QRS_NEXT_CUT()
PTP {E1 36177.176,E2 36177.176}
PTP {X 0,Y 759.945,A -85,B 0,C 180,E1 36177.176,E2 36177.176,E3 0,E4 0,E5 0,E6 0}
QRS_SPEED_INIT()
LIN {X 0,Y 759.945,Z 1215,A -85,B 0,C 180,E1 36177.176,E2 36177.176,E3 0,E4 0,E5 0,E6 0} C_VEL
LIN {X 0,Y 759.945,Z 319.648,A -85,B 0,C 180,E1 36177.176,E2 36177.176} C_VEL
LIN {X 0,Y 759.945,Z 311.576,A -85,B 0,C 180,E1 36177.176,E2 36177.176} C_VEL
LIN {X 0,Y 759.914,Z 309.576,A -85,B 0,C 180,E1 36177.025,E2 36177.025} C_VEL
LIN {X 0,Y 759.839,Z 309.574,A -85,B 0,C 180,E1 36174.336,E2 36174.336} C_VEL
LIN {X 0,Y 759.839,Z 309.572,A -85,B 0,C 180,E1 36171.906,E2 36171.906} C_VEL
LIN {X 0,Y 759.916,Z 309.571,A -85,B 0,C 180,E1 36169.155,E2 36169.155} C_VEL
LIN {X 0,Y 759.839,Z 309.575,A -85,B 0,C 180,E1 36166.298,E2 36166.298} C_VEL
LIN {X 0,Y 759.826,Z 309.574,A -85,B 0,C 180,E1 36163.957,E2 36163.957} C_VEL
LIN {X 0,Y 759.829,Z 309.574,A -85,B 0,C 180,E1 36161.669,E2 36161.669} C_VEL
LIN {X 0,Y 759.912,Z 309.571,A -85,B 0,C 180,E1 36158.948,E2 36158.948} C_VEL
LIN {X 0,Y 759.831,Z 309.576,A -85,B 0,C 180,E1 36156.089,E2 36156.089} C_VEL
LIN {X 0,Y 759.817,Z 309.575,A -85,B 0,C 180,E1 36153.825,E2 36153.825} C_VEL
LIN {X 0,Y 759.814,Z 309.576,A -85,B 0,C 180,E1 36151.551,E2 36151.551} C_VEL
LIN {X 0,Y 759.828,Z 309.575,A -85,B 0,C 180,E1 36149.209,E2 36149.209} C_VEL
LIN {X 0,Y 759.89,Z 309.576,A -85,B 0,C 180,E1 36146.36,E2 36146.36} C_VEL
LIN {X 0,Y 759.815,Z 309.577,A -85,B 0,C 180,E1 36143.771,E2 36143.771} C_VEL
LIN {X 0,Y 759.802,Z 309.576,A -85,B 0,C 180,E1 36141.504,E2 36141.504} C_VEL
LIN {X 0,Y 759.801,Z 309.578,A -85,B 0,C 180,E1 36139.252,E2 36139.252} C_VEL
LIN {X 0,Y 759.811,Z 309.578,A -85,B 0,C 180,E1 36137.025,E2 36137.025} C_VEL
LIN {X 0,Y 759.909,Z 309.578,A -85,B 0,C 180,E1 36134.291,E2 36134.291} C_VEL
LIN {X 0,Y 759.83,Z 309.76,A -85,B 0,C 180,E1 36131.629,E2 36131.629} C_VEL
LIN {X 0,Y 759.819,Z 321.429,A -85,B 0,C 180,E1 36130.869,E2 36130.869} C_VEL
LIN {X 0,Y 759.897,Z 497.056,A -85,B 0,C 180,E1 36128.746,E2 36128.746} C_VEL
LIN {X 0,Y 759.916,Z 717.097,A -85,B 0,C 180,E1 36126.177,E2 36126.177} C_VEL
LIN {X 0,Y 759.91,Z 798.77,A -85,B 0,C 180,E1 36125.223,E2 36125.223} C_VEL
LIN {X 0,Y 759.911,Z 825.377,A -85,B 0,C 180,E1 36124.77,E2 36124.77} C_VEL
LIN {X 0,Y 759.914,Z 852.595,A -85,B 0,C 180,E1 36124.143,E2 36124.143} C_VEL
LIN {X 0,Y 759.907,Z 874.72,A -85,B 0,C 180,E1 36123.506,E2 36123.506} C_VEL
LIN {X 0,Y 759.919,Z 892.583,A -85,B 0,C 180,E1 36122.915,E2 36122.915} C_VEL
LIN {X 0,Y 759.919,Z 911.329,A -85,B 0,C 180,E1 36122.215,E2 36122.215} C_VEL
LIN {X 0,Y 759.913,Z 929.676,A -85,B 0,C 180,E1 36121.446,E2 36121.446} C_VEL
LIN {X 0,Y 759.915,Z 948.5,A -85,B 0,C 180,E1 36120.566,E2 36120.566} C_VEL
LIN {X 0,Y 759.911,Z 966.95,A -85,B 0,C 180,E1 36119.611,E2 36119.611} C_VEL
LIN {X 0,Y 759.909,Z 986.655,A -85,B 0,C 180,E1 36118.483,E2 36118.483} C_VEL
LIN {X 0,Y 759.91,Z 1010.382,A -85,B 0,C 180,E1 36116.954,E2 36116.954} C_VEL
LIN {X 0,Y 759.915,Z 1028.464,A -85,B 0,C 180,E1 36115.65,E2 36115.65} C_VEL
LIN {X 0,Y 759.893,Z 1046.844,A -85,B 0,C 180,E1 36114.195,E2 36114.195} C_VEL
LIN {X 0,Y 759.92,Z 1065.796,A -85,B 0,C 180,E1 36112.512,E2 36112.512} C_VEL
LIN {X 0,Y 759.897,Z 1080.62,A -85,B 0,C 180,E1 36111.052,E2 36111.052} C_VEL
LIN {X 0,Y 759.914,Z 1094.69,A -85,B 0,C 180,E1 36109.524,E2 36109.524} C_VEL
LIN {X 0,Y 759.9,Z 1109.841,A -85,B 0,C 180,E1 36107.695,E2 36107.695} C_VEL
LIN {X 0,Y 759.89,Z 1122.953,A -85,B 0,C 180,E1 36105.871,E2 36105.871} C_VEL
LIN {X 0,Y 759.917,Z 1132.856,A -85,B 0,C 180,E1 36104.321,E2 36104.321} C_VEL
LIN {X 0,Y 759.908,Z 1141.641,A -85,B 0,C 180,E1 36102.771,E2 36102.771} C_VEL
LIN {X 0,Y 759.903,Z 1149.647,A -85,B 0,C 180,E1 36101.152,E2 36101.152} C_VEL
LIN {X 0,Y 759.916,Z 1157.473,A -85,B 0,C 180,E1 36099.303,E2 36099.303} C_VEL
LIN {X 0,Y 759.91,Z 1164.123,A -85,B 0,C 180,E1 36097.333,E2 36097.333} C_VEL
LIN {X 0,Y 759.906,Z 1169.35,A -85,B 0,C 180,E1 36095.285,E2 36095.285} C_VEL
LIN {X 0,Y 759.909,Z 1172.83,A -85,B 0,C 180,E1 36093.243,E2 36093.243} C_VEL
LIN {X 0,Y 759.911,Z 1174.612,A -85,B 0,C 180,E1 36091.282,E2 36091.282} C_VEL
LIN {X 0,Y 759.889,Z 1174.863,A -85,B 0,C 180,E1 36089.472,E2 36089.472} C_VEL
LIN {X 0,Y 759.907,Z 1173.954,A -85,B 0,C 180,E1 36087.662,E2 36087.662} C_VEL
LIN {X 0,Y 759.909,Z 1171.128,A -85,B 0,C 180,E1 36085.548,E2 36085.548} C_VEL
LIN {X 0,Y 759.918,Z 1166.878,A -85,B 0,C 180,E1 36083.579,E2 36083.579} C_VEL
LIN {X 0,Y 759.916,Z 1160.788,A -85,B 0,C 180,E1 36081.526,E2 36081.526} C_VEL
LIN {X 0,Y 759.893,Z 1152.605,A -85,B 0,C 180,E1 36079.399,E2 36079.399} C_VEL
LIN {X 0,Y 759.913,Z 1142.939,A -85,B 0,C 180,E1 36077.384,E2 36077.384} C_VEL
LIN {X 0,Y 759.918,Z 1133.86,A -85,B 0,C 180,E1 36075.756,E2 36075.756} C_VEL
LIN {X 0,Y 759.894,Z 1123.989,A -85,B 0,C 180,E1 36074.195,E2 36074.195} C_VEL
LIN {X 0,Y 759.908,Z 1112.833,A -85,B 0,C 180,E1 36072.622,E2 36072.622} C_VEL
LIN {X 0,Y 759.912,Z 1097.622,A -85,B 0,C 180,E1 36070.716,E2 36070.716} C_VEL
LIN {X 0,Y 759.893,Z 1082.269,A -85,B 0,C 180,E1 36069.029,E2 36069.029} C_VEL
LIN {X 0,Y 759.903,Z 1067.592,A -85,B 0,C 180,E1 36067.569,E2 36067.569} C_VEL
LIN {X 0,Y 759.892,Z 1048.945,A -85,B 0,C 180,E1 36065.886,E2 36065.886} C_VEL
LIN {X 0,Y 759.917,Z 1029.425,A -85,B 0,C 180,E1 36064.332,E2 36064.332} C_VEL
LIN {X 0,Y 759.91,Z 1012.274,A -85,B 0,C 180,E1 36063.088,E2 36063.088} C_VEL
LIN {X 0,Y 759.915,Z 990.289,A -85,B 0,C 180,E1 36061.642,E2 36061.642} C_VEL
LIN {X 0,Y 759.908,Z 967.865,A -85,B 0,C 180,E1 36060.348,E2 36060.348} C_VEL
LIN {X 0,Y 759.917,Z 949.16,A -85,B 0,C 180,E1 36059.376,E2 36059.376} C_VEL
LIN {X 0,Y 759.913,Z 930.486,A -85,B 0,C 180,E1 36058.5,E2 36058.5} C_VEL
LIN {X 0,Y 759.919,Z 911.728,A -85,B 0,C 180,E1 36057.711,E2 36057.711} C_VEL
LIN {X 0,Y 759.92,Z 893.856,A -85,B 0,C 180,E1 36057.04,E2 36057.04} C_VEL
LIN {X 0,Y 759.909,Z 875.417,A -85,B 0,C 180,E1 36056.426,E2 36056.426} C_VEL
LIN {X 0,Y 759.912,Z 853.71,A -85,B 0,C 180,E1 36055.795,E2 36055.795} C_VEL
LIN {X 0,Y 759.914,Z 826.054,A -85,B 0,C 180,E1 36055.155,E2 36055.155} C_VEL
LIN {X 0,Y 759.91,Z 799.959,A -85,B 0,C 180,E1 36054.704,E2 36054.704} C_VEL
LIN {X 0,Y 759.919,Z 743.099,A -85,B 0,C 180,E1 36054.031,E2 36054.031} C_VEL
LIN {X 0,Y 759.91,Z 519.207,A -85,B 0,C 180,E1 36051.428,E2 36051.428} C_VEL
LIN {X 0,Y 759.834,Z 329.757,A -85,B 0,C 180,E1 36049.144,E2 36049.144} C_VEL
LIN {X 0,Y 759.825,Z 320.904,A -85,B 0,C 180,E1 36049.031,E2 36049.031} C_VEL
LIN {X 0,Y 759.848,Z 309.579,A -85,B 0,C 180,E1 36048.254,E2 36048.254} C_VEL
LIN {X 0,Y 759.842,Z 309.577,A -85,B 0,C 180,E1 36045.177,E2 36045.177} C_VEL
LIN {X 0,Y 759.817,Z 309.577,A -85,B 0,C 180,E1 36042.864,E2 36042.864} C_VEL
LIN {X 0,Y 759.808,Z 309.577,A -85,B 0,C 180,E1 36040.648,E2 36040.648} C_VEL
LIN {X 0,Y 759.805,Z 309.577,A -85,B 0,C 180,E1 36038.466,E2 36038.466} C_VEL
LIN {X 0,Y 759.82,Z 309.577,A -85,B 0,C 180,E1 36036.102,E2 36036.102} C_VEL
LIN {X 0,Y 759.886,Z 309.578,A -85,B 0,C 180,E1 36033.279,E2 36033.279} C_VEL
LIN {X 0,Y 759.815,Z 309.576,A -85,B 0,C 180,E1 36030.704,E2 36030.704} C_VEL
LIN {X 0,Y 759.807,Z 309.577,A -85,B 0,C 180,E1 36028.45,E2 36028.45} C_VEL
LIN {X 0,Y 759.807,Z 309.576,A -85,B 0,C 180,E1 36026.243,E2 36026.243} C_VEL
LIN {X 0,Y 759.814,Z 309.576,A -85,B 0,C 180,E1 36024.042,E2 36024.042} C_VEL
LIN {X 0,Y 759.862,Z 309.577,A -85,B 0,C 180,E1 36021.519,E2 36021.519} C_VEL
LIN {X 0,Y 759.844,Z 309.574,A -85,B 0,C 180,E1 36018.569,E2 36018.569} C_VEL
LIN {X 0,Y 759.822,Z 309.574,A -85,B 0,C 180,E1 36016.2,E2 36016.2} C_VEL
LIN {X 0,Y 759.822,Z 309.574,A -85,B 0,C 180,E1 36013.935,E2 36013.935} C_VEL
LIN {X 0,Y 759.843,Z 309.576,A -85,B 0,C 180,E1 36011.538,E2 36011.538} C_VEL
LIN {X 0,Y 759.897,Z 309.571,A -85,B 0,C 180,E1 36008.627,E2 36008.627} C_VEL
LIN {X 0,Y 759.837,Z 309.573,A -85,B 0,C 180,E1 36006.043,E2 36006.043} C_VEL
LIN {X 0,Y 759.833,Z 309.573,A -85,B 0,C 180,E1 36003.697,E2 36003.697} C_VEL
LIN {X 0,Y 759.865,Z 309.575,A -85,B 0,C 180,E1 36001.206,E2 36001.206} C_VEL
LIN {X 0,Y 759.867,Z 309.57,A -85,B 0,C 180,E1 35998.115,E2 35998.115} C_VEL
LIN {X 0,Y 759.842,Z 309.572,A -85,B 0,C 180,E1 35995.623,E2 35995.623} C_VEL
LIN {X 0,Y 759.863,Z 309.575,A -85,B 0,C 180,E1 35993.123,E2 35993.123} C_VEL
LIN {X 0,Y 759.906,Z 309.567,A -85,B 0,C 180,E1 35990.151,E2 35990.151} C_VEL
LIN {X 0,Y 759.85,Z 309.572,A -85,B 0,C 180,E1 35987.46,E2 35987.46} C_VEL
LIN {X 0,Y 759.875,Z 309.574,A -85,B 0,C 180,E1 35984.898,E2 35984.898} C_VEL
LIN {X 0,Y 759.904,Z 309.567,A -85,B 0,C 180,E1 35981.909,E2 35981.909} C_VEL
LIN {X 0,Y 759.858,Z 309.57,A -85,B 0,C 180,E1 35979.269,E2 35979.269} C_VEL
LIN {X 0,Y 759.895,Z 309.577,A -85,B 0,C 180,E1 35976.585,E2 35976.585} C_VEL
LIN {X 0,Y 759.894,Z 309.566,A -85,B 0,C 180,E1 35973.593,E2 35973.593} C_VEL
LIN {X 0,Y 759.867,Z 309.572,A -85,B 0,C 180,E1 35970.864,E2 35970.864} C_VEL
LIN {X 0,Y 759.911,Z 309.575,A -85,B 0,C 180,E1 35968.154,E2 35968.154} C_VEL
LIN {X 0,Y 759.887,Z 309.567,A -85,B 0,C 180,E1 35965.266,E2 35965.266} C_VEL
LIN {X 0,Y 759.887,Z 309.574,A -85,B 0,C 180,E1 35962.466,E2 35962.466} C_VEL
LIN {X 0,Y 759.91,Z 309.566,A -85,B 0,C 180,E1 35959.509,E2 35959.509} C_VEL
LIN {X 0,Y 759.876,Z 309.571,A -85,B 0,C 180,E1 35956.72,E2 35956.72} C_VEL
LIN {X 0,Y 759.913,Z 309.577,A -85,B 0,C 180,E1 35953.967,E2 35953.967} C_VEL
LIN {X 0,Y 759.9,Z 309.834,A -85,B 0,C 180,E1 35953.53,E2 35953.53} C_VEL
LIN {X 0,Y 759.904,Z 350.585,A -85,B 0,C 180,E1 35950.919,E2 35950.919} C_VEL
LIN {X 0,Y 759.912,Z 566.438,A -85,B 0,C 180,E1 35948.324,E2 35948.324} C_VEL
LIN {X 0,Y 759.917,Z 792.185,A -85,B 0,C 180,E1 35945.706,E2 35945.706} C_VEL
LIN {X 0,Y 759.911,Z 831.844,A -85,B 0,C 180,E1 35945.223,E2 35945.223} C_VEL
LIN {X 0,Y 759.908,Z 857.526,A -85,B 0,C 180,E1 35944.77,E2 35944.77} C_VEL
LIN {X 0,Y 759.913,Z 884.353,A -85,B 0,C 180,E1 35944.143,E2 35944.143} C_VEL
LIN {X 0,Y 759.907,Z 909.243,A -85,B 0,C 180,E1 35943.411,E2 35943.411} C_VEL
LIN {X 0,Y 759.918,Z 937.245,A -85,B 0,C 180,E1 35942.423,E2 35942.423} C_VEL
LIN {X 0,Y 759.915,Z 958.588,A -85,B 0,C 180,E1 35941.539,E2 35941.539} C_VEL
LIN {X 0,Y 759.912,Z 977.503,A -85,B 0,C 180,E1 35940.661,E2 35940.661} C_VEL
LIN {X 0,Y 759.913,Z 995.702,A -85,B 0,C 180,E1 35939.723,E2 35939.723} C_VEL
LIN {X 0,Y 759.909,Z 1013.707,A -85,B 0,C 180,E1 35938.702,E2 35938.702} C_VEL
LIN {X 0,Y 759.911,Z 1035.516,A -85,B 0,C 180,E1 35937.335,E2 35937.335} C_VEL
LIN {X 0,Y 759.912,Z 1056.845,A -85,B 0,C 180,E1 35935.818,E2 35935.818} C_VEL
LIN {X 0,Y 759.91,Z 1073.823,A -85,B 0,C 180,E1 35934.485,E2 35934.485} C_VEL
LIN {X 0,Y 759.901,Z 1092.853,A -85,B 0,C 180,E1 35932.84,E2 35932.84} C_VEL
LIN {X 0,Y 759.895,Z 1109.495,A -85,B 0,C 180,E1 35931.213,E2 35931.213} C_VEL
LIN {X 0,Y 759.905,Z 1122.958,A -85,B 0,C 180,E1 35929.764,E2 35929.764} C_VEL
LIN {X 0,Y 759.897,Z 1135.732,A -85,B 0,C 180,E1 35928.249,E2 35928.249} C_VEL
LIN {X 0,Y 759.909,Z 1150.031,A -85,B 0,C 180,E1 35926.354,E2 35926.354} C_VEL
LIN {X 0,Y 759.909,Z 1162.194,A -85,B 0,C 180,E1 35924.477,E2 35924.477} C_VEL
LIN {X 0,Y 759.91,Z 1171.058,A -85,B 0,C 180,E1 35922.925,E2 35922.925} C_VEL
LIN {X 0,Y 759.91,Z 1178.784,A -85,B 0,C 180,E1 35921.383,E2 35921.383} C_VEL
LIN {X 0,Y 759.906,Z 1186.43,A -85,B 0,C 180,E1 35919.619,E2 35919.619} C_VEL
LIN {X 0,Y 759.908,Z 1193.594,A -85,B 0,C 180,E1 35917.561,E2 35917.561} C_VEL
LIN {X 0,Y 759.91,Z 1199.108,A -85,B 0,C 180,E1 35915.436,E2 35915.436} C_VEL
LIN {X 0,Y 759.916,Z 1202.585,A -85,B 0,C 180,E1 35913.47,E2 35913.47} C_VEL
LIN {X 0,Y 759.914,Z 1204.58,A -85,B 0,C 180,E1 35911.432,E2 35911.432} C_VEL
LIN {X 0,Y 759.889,Z 1204.849,A -85,B 0,C 180,E1 35909.472,E2 35909.472} C_VEL
LIN {X 0,Y 759.907,Z 1203.907,A -85,B 0,C 180,E1 35907.662,E2 35907.662} C_VEL
LIN {X 0,Y 759.908,Z 1201.054,A -85,B 0,C 180,E1 35905.548,E2 35905.548} C_VEL
LIN {X 0,Y 759.914,Z 1196.566,A -85,B 0,C 180,E1 35903.503,E2 35903.503} C_VEL
LIN {X 0,Y 759.913,Z 1190.629,A -85,B 0,C 180,E1 35901.526,E2 35901.526} C_VEL
LIN {X 0,Y 759.896,Z 1182.68,A -85,B 0,C 180,E1 35899.462,E2 35899.462} C_VEL
LIN {X 0,Y 759.905,Z 1173.111,A -85,B 0,C 180,E1 35897.461,E2 35897.461} C_VEL
LIN {X 0,Y 759.91,Z 1164.056,A -85,B 0,C 180,E1 35895.834,E2 35895.834} C_VEL
LIN {X 0,Y 759.894,Z 1154.212,A -85,B 0,C 180,E1 35894.273,E2 35894.273} C_VEL
LIN {X 0,Y 759.904,Z 1143.666,A -85,B 0,C 180,E1 35892.78,E2 35892.78} C_VEL
LIN {X 0,Y 759.896,Z 1130.456,A -85,B 0,C 180,E1 35891.1,E2 35891.1} C_VEL
LIN {X 0,Y 759.898,Z 1113.394,A -85,B 0,C 180,E1 35889.191,E2 35889.191} C_VEL
LIN {X 0,Y 759.898,Z 1098.828,A -85,B 0,C 180,E1 35887.732,E2 35887.732} C_VEL
LIN {X 0,Y 759.911,Z 1082.654,A -85,B 0,C 180,E1 35886.258,E2 35886.258} C_VEL
LIN {X 0,Y 759.91,Z 1061.274,A -85,B 0,C 180,E1 35884.516,E2 35884.516} C_VEL
LIN {X 0,Y 759.91,Z 1044.049,A -85,B 0,C 180,E1 35883.257,E2 35883.257} C_VEL
LIN {X 0,Y 759.914,Z 1026.242,A -85,B 0,C 180,E1 35882.069,E2 35882.069} C_VEL
LIN {X 0,Y 759.905,Z 1003.454,A -85,B 0,C 180,E1 35880.695,E2 35880.695} C_VEL
LIN {X 0,Y 759.916,Z 981.266,A -85,B 0,C 180,E1 35879.525,E2 35879.525} C_VEL
LIN {X 0,Y 759.912,Z 961.681,A -85,B 0,C 180,E1 35878.598,E2 35878.598} C_VEL
LIN {X 0,Y 759.918,Z 942.461,A -85,B 0,C 180,E1 35877.785,E2 35877.785} C_VEL
LIN {X 0,Y 759.919,Z 923.853,A -85,B 0,C 180,E1 35877.085,E2 35877.085} C_VEL
LIN {X 0,Y 759.909,Z 905.51,A -85,B 0,C 180,E1 35876.474,E2 35876.474} C_VEL
LIN {X 0,Y 759.913,Z 882.835,A -85,B 0,C 180,E1 35875.818,E2 35875.818} C_VEL
LIN {X 0,Y 759.911,Z 855.67,A -85,B 0,C 180,E1 35875.191,E2 35875.191} C_VEL
LIN {X 0,Y 759.91,Z 829.101,A -85,B 0,C 180,E1 35874.737,E2 35874.737} C_VEL
LIN {X 0,Y 759.915,Z 735.994,A -85,B 0,C 180,E1 35873.651,E2 35873.651} C_VEL
LIN {X 0,Y 759.912,Z 513.174,A -85,B 0,C 180,E1 35871.045,E2 35871.045} C_VEL
LIN {X 0,Y 759.904,Z 350.467,A -85,B 0,C 180,E1 35869.074,E2 35869.074} C_VEL
LIN {X 0,Y 759.9,Z 309.834,A -85,B 0,C 180,E1 35866.47,E2 35866.47} C_VEL
LIN {X 0,Y 759.913,Z 309.577,A -85,B 0,C 180,E1 35866.033,E2 35866.033} C_VEL
LIN {X 0,Y 759.877,Z 309.57,A -85,B 0,C 180,E1 35863.201,E2 35863.201} C_VEL
LIN {X 0,Y 759.907,Z 309.566,A -85,B 0,C 180,E1 35860.443,E2 35860.443} C_VEL
LIN {X 0,Y 759.887,Z 309.575,A -85,B 0,C 180,E1 35857.534,E2 35857.534} C_VEL
LIN {X 0,Y 759.892,Z 309.566,A -85,B 0,C 180,E1 35854.678,E2 35854.678} C_VEL
LIN {X 0,Y 759.908,Z 309.578,A -85,B 0,C 180,E1 35851.669,E2 35851.669} C_VEL
LIN {X 0,Y 759.865,Z 309.571,A -85,B 0,C 180,E1 35848.952,E2 35848.952} C_VEL
LIN {X 0,Y 759.911,Z 309.566,A -85,B 0,C 180,E1 35846.189,E2 35846.189} C_VEL
LIN {X 0,Y 759.882,Z 309.575,A -85,B 0,C 180,E1 35843.251,E2 35843.251} C_VEL
LIN {X 0,Y 759.864,Z 309.569,A -85,B 0,C 180,E1 35840.569,E2 35840.569} C_VEL
LIN {X 0,Y 759.91,Z 309.57,A -85,B 0,C 180,E1 35837.774,E2 35837.774} C_VEL
LIN {X 0,Y 759.865,Z 309.573,A -85,B 0,C 180,E1 35834.946,E2 35834.946} C_VEL
LIN {X 0,Y 759.862,Z 309.57,A -85,B 0,C 180,E1 35832.308,E2 35832.308} C_VEL
LIN {X 0,Y 759.913,Z 309.573,A -85,B 0,C 180,E1 35829.467,E2 35829.467} C_VEL
LIN {X 0,Y 759.856,Z 309.574,A -85,B 0,C 180,E1 35826.726,E2 35826.726} C_VEL
LIN {X 0,Y 759.849,Z 309.571,A -85,B 0,C 180,E1 35824.226,E2 35824.226} C_VEL
LIN {X 0,Y 759.915,Z 309.568,A -85,B 0,C 180,E1 35821.508,E2 35821.508} C_VEL
LIN {X 0,Y 759.856,Z 309.574,A -85,B 0,C 180,E1 35818.643,E2 35818.643} C_VEL
LIN {X 0,Y 759.914,Z 309.576,A -85,B 0,C 180,E1 35817.025,E2 35817.025} C_VEL
LIN {X 0,Y 758.859,Z 309.699,A -85,B 0,C 180,E1 35816.444,E2 35816.444} C_VEL
LIN {X 0,Y 752.447,Z 310.504,A -85,B 0,C 180,E1 35814.818,E2 35814.818} C_VEL
LIN {X 0,Y 751.904,Z 310.564,A -85,B 0,C 180,E1 35814.396,E2 35814.396} C_VEL
LIN {X 0,Y 751.897,Z 310.561,A -85,B 0,C 180,E1 35811.973,E2 35811.973} C_VEL
LIN {X 0,Y 751.966,Z 310.558,A -85,B 0,C 180,E1 35809.271,E2 35809.271} C_VEL
LIN {X 0,Y 751.908,Z 310.563,A -85,B 0,C 180,E1 35806.386,E2 35806.386} C_VEL
LIN {X 0,Y 751.888,Z 310.563,A -85,B 0,C 180,E1 35804.021,E2 35804.021} C_VEL
LIN {X 0,Y 751.889,Z 310.563,A -85,B 0,C 180,E1 35801.708,E2 35801.708} C_VEL
LIN {X 0,Y 751.955,Z 310.559,A -85,B 0,C 180,E1 35799.041,E2 35799.041} C_VEL
LIN {X 0,Y 751.898,Z 310.565,A -85,B 0,C 180,E1 35796.155,E2 35796.155} C_VEL
LIN {X 0,Y 751.877,Z 310.564,A -85,B 0,C 180,E1 35793.799,E2 35793.799} C_VEL
LIN {X 0,Y 751.876,Z 310.565,A -85,B 0,C 180,E1 35791.523,E2 35791.523} C_VEL
LIN {X 0,Y 751.898,Z 310.562,A -85,B 0,C 180,E1 35789.115,E2 35789.115} C_VEL
LIN {X 0,Y 751.9,Z 310.564,A -85,B 0,C 180,E1 35786.046,E2 35786.046} C_VEL
LIN {X 0,Y 751.871,Z 310.567,A -85,B 0,C 180,E1 35783.695,E2 35783.695} C_VEL
LIN {X 0,Y 751.862,Z 310.564,A -85,B 0,C 180,E1 35781.439,E2 35781.439} C_VEL
LIN {X 0,Y 751.867,Z 310.567,A -85,B 0,C 180,E1 35779.133,E2 35779.133} C_VEL
LIN {X 0,Y 751.93,Z 310.567,A -85,B 0,C 180,E1 35776.554,E2 35776.554} C_VEL
LIN {X 0,Y 751.886,Z 310.569,A -85,B 0,C 180,E1 35773.643,E2 35773.643} C_VEL
LIN {X 0,Y 751.978,Z 310.677,A -85,B 0,C 180,E1 35772.101,E2 35772.101} C_VEL
LIN {X 0,Y 753.147,Z 314.7,A -85,B 0,C 180,E1 35771.744,E2 35771.744} C_VEL
LIN {X 0,Y 753.251,Z 321.517,A -85,B 0,C 180,E1 35771.302,E2 35771.302} C_VEL
LIN {X 0,Y 753.757,Z 324.477,A -85,B 0,C 180,E1 35771.232,E2 35771.232} C_VEL
LIN {X 0,Y 753.644,Z 503.901,A -85,B 0,C 180,E1 35769.047,E2 35769.047} C_VEL
LIN {X 0,Y 753.443,Z 729.229,A -85,B 0,C 180,E1 35766.397,E2 35766.397} C_VEL
LIN {X 0,Y 753.353,Z 799.594,A -85,B 0,C 180,E1 35765.564,E2 35765.564} C_VEL
LIN {X 0,Y 753.277,Z 826.438,A -85,B 0,C 180,E1 35765.099,E2 35765.099} C_VEL
LIN {X 0,Y 753.196,Z 853.912,A -85,B 0,C 180,E1 35764.457,E2 35764.457} C_VEL
LIN {X 0,Y 753.096,Z 877.658,A -85,B 0,C 180,E1 35763.758,E2 35763.758} C_VEL
LIN {X 0,Y 753.006,Z 902.747,A -85,B 0,C 180,E1 35762.893,E2 35762.893} C_VEL
LIN {X 0,Y 752.86,Z 927.706,A -85,B 0,C 180,E1 35761.864,E2 35761.864} C_VEL
LIN {X 0,Y 752.761,Z 947.625,A -85,B 0,C 180,E1 35760.933,E2 35760.933} C_VEL
LIN {X 0,Y 752.667,Z 966.211,A -85,B 0,C 180,E1 35759.966,E2 35759.966} C_VEL
LIN {X 0,Y 752.574,Z 984.97,A -85,B 0,C 180,E1 35758.888,E2 35758.888} C_VEL
LIN {X 0,Y 752.438,Z 1007.964,A -85,B 0,C 180,E1 35757.416,E2 35757.416} C_VEL
LIN {X 0,Y 752.339,Z 1027.364,A -85,B 0,C 180,E1 35756.013,E2 35756.013} C_VEL
LIN {X 0,Y 752.28,Z 1044.293,A -85,B 0,C 180,E1 35754.667,E2 35754.667} C_VEL
LIN {X 0,Y 752.173,Z 1063.244,A -85,B 0,C 180,E1 35753.005,E2 35753.005} C_VEL
LIN {X 0,Y 752.11,Z 1079.847,A -85,B 0,C 180,E1 35751.362,E2 35751.362} C_VEL
LIN {X 0,Y 752.054,Z 1093.276,A -85,B 0,C 180,E1 35749.898,E2 35749.898} C_VEL
LIN {X 0,Y 752.028,Z 1106.421,A -85,B 0,C 180,E1 35748.317,E2 35748.317} C_VEL
LIN {X 0,Y 751.966,Z 1121.591,A -85,B 0,C 180,E1 35746.25,E2 35746.25} C_VEL
LIN {X 0,Y 751.955,Z 1132.578,A -85,B 0,C 180,E1 35744.524,E2 35744.524} C_VEL
LIN {X 0,Y 751.926,Z 1141.644,A -85,B 0,C 180,E1 35742.908,E2 35742.908} C_VEL
LIN {X 0,Y 751.93,Z 1149.293,A -85,B 0,C 180,E1 35741.35,E2 35741.35} C_VEL
LIN {X 0,Y 751.915,Z 1156.846,A -85,B 0,C 180,E1 35739.568,E2 35739.568} C_VEL
LIN {X 0,Y 751.912,Z 1163.685,A -85,B 0,C 180,E1 35737.565,E2 35737.565} C_VEL
LIN {X 0,Y 751.909,Z 1169.179,A -85,B 0,C 180,E1 35735.418,E2 35735.418} C_VEL
LIN {X 0,Y 751.91,Z 1172.729,A -85,B 0,C 180,E1 35733.354,E2 35733.354} C_VEL
LIN {X 0,Y 751.912,Z 1174.589,A -85,B 0,C 180,E1 35731.372,E2 35731.372} C_VEL
LIN {X 0,Y 751.889,Z 1174.863,A -85,B 0,C 180,E1 35729.467,E2 35729.467} C_VEL
LIN {X 0,Y 751.907,Z 1173.953,A -85,B 0,C 180,E1 35727.637,E2 35727.637} C_VEL
LIN {X 0,Y 751.907,Z 1171.127,A -85,B 0,C 180,E1 35725.5,E2 35725.5} C_VEL
LIN {X 0,Y 751.917,Z 1166.876,A -85,B 0,C 180,E1 35723.51,E2 35723.51} C_VEL
LIN {X 0,Y 751.923,Z 1160.786,A -85,B 0,C 180,E1 35721.435,E2 35721.435} C_VEL
LIN {X 0,Y 751.904,Z 1152.823,A -85,B 0,C 180,E1 35719.338,E2 35719.338} C_VEL
LIN {X 0,Y 751.941,Z 1143.349,A -85,B 0,C 180,E1 35717.326,E2 35717.326} C_VEL
LIN {X 0,Y 751.961,Z 1134.324,A -85,B 0,C 180,E1 35715.681,E2 35715.681} C_VEL
LIN {X 0,Y 751.957,Z 1124.51,A -85,B 0,C 180,E1 35714.103,E2 35714.103} C_VEL
LIN {X 0,Y 751.998,Z 1113.996,A -85,B 0,C 180,E1 35712.593,E2 35712.593} C_VEL
LIN {X 0,Y 752.032,Z 1101.41,A -85,B 0,C 180,E1 35710.969,E2 35710.969} C_VEL
LIN {X 0,Y 752.09,Z 1083.741,A -85,B 0,C 180,E1 35708.956,E2 35708.956} C_VEL
LIN {X 0,Y 752.152,Z 1069.295,A -85,B 0,C 180,E1 35707.49,E2 35707.49} C_VEL
LIN {X 0,Y 752.212,Z 1053.624,A -85,B 0,C 180,E1 35706.041,E2 35706.041} C_VEL
LIN {X 0,Y 752.335,Z 1032.971,A -85,B 0,C 180,E1 35704.326,E2 35704.326} C_VEL
LIN {X 0,Y 752.414,Z 1014.687,A -85,B 0,C 180,E1 35702.969,E2 35702.969} C_VEL
LIN {X 0,Y 752.492,Z 996.808,A -85,B 0,C 180,E1 35701.761,E2 35701.761} C_VEL
LIN {X 0,Y 752.629,Z 974.253,A -85,B 0,C 180,E1 35700.383,E2 35700.383} C_VEL
LIN {X 0,Y 752.753,Z 951.212,A -85,B 0,C 180,E1 35699.156,E2 35699.156} C_VEL
LIN {X 0,Y 752.846,Z 931.449,A -85,B 0,C 180,E1 35698.214,E2 35698.214} C_VEL
LIN {X 0,Y 752.943,Z 912.835,A -85,B 0,C 180,E1 35697.42,E2 35697.42} C_VEL
LIN {X 0,Y 753.031,Z 893.843,A -85,B 0,C 180,E1 35696.699,E2 35696.699} C_VEL
LIN {X 0,Y 753.107,Z 874.824,A -85,B 0,C 180,E1 35696.064,E2 35696.064} C_VEL
LIN {X 0,Y 753.201,Z 852.326,A -85,B 0,C 180,E1 35695.412,E2 35695.412} C_VEL
LIN {X 0,Y 753.295,Z 825.342,A -85,B 0,C 180,E1 35694.789,E2 35694.789} C_VEL
LIN {X 0,Y 753.353,Z 797.608,A -85,B 0,C 180,E1 35694.317,E2 35694.317} C_VEL
LIN {X 0,Y 753.612,Z 550.858,A -85,B 0,C 180,E1 35691.424,E2 35691.424} C_VEL
LIN {X 0,Y 753.769,Z 349.831,A -85,B 0,C 180,E1 35688.993,E2 35688.993} C_VEL
LIN {X 0,Y 753.581,Z 322.693,A -85,B 0,C 180,E1 35688.645,E2 35688.645} C_VEL
LIN {X 0,Y 753.124,Z 320.521,A -85,B 0,C 180,E1 35688.562,E2 35688.562} C_VEL
LIN {X 0,Y 753.082,Z 313.814,A -85,B 0,C 180,E1 35688.101,E2 35688.101} C_VEL
LIN {X 0,Y 751.974,Z 310.566,A -85,B 0,C 180,E1 35687.786,E2 35687.786} C_VEL
LIN {X 0,Y 751.888,Z 310.567,A -85,B 0,C 180,E1 35685.03,E2 35685.03} C_VEL
LIN {X 0,Y 751.873,Z 310.566,A -85,B 0,C 180,E1 35682.706,E2 35682.706} C_VEL
LIN {X 0,Y 751.871,Z 310.567,A -85,B 0,C 180,E1 35680.465,E2 35680.465} C_VEL
LIN {X 0,Y 751.888,Z 310.566,A -85,B 0,C 180,E1 35678.101,E2 35678.101} C_VEL
LIN {X 0,Y 751.916,Z 310.564,A -85,B 0,C 180,E1 35675.136,E2 35675.136} C_VEL
LIN {X 0,Y 751.868,Z 310.567,A -85,B 0,C 180,E1 35672.671,E2 35672.671} C_VEL
LIN {X 0,Y 751.864,Z 310.564,A -85,B 0,C 180,E1 35670.443,E2 35670.443} C_VEL
LIN {X 0,Y 751.866,Z 310.566,A -85,B 0,C 180,E1 35668.258,E2 35668.258} C_VEL
LIN {X 0,Y 751.881,Z 310.565,A -85,B 0,C 180,E1 35665.946,E2 35665.946} C_VEL
LIN {X 0,Y 751.975,Z 310.565,A -85,B 0,C 180,E1 35663.178,E2 35663.178} C_VEL
LIN {X 0,Y 751.889,Z 310.561,A -85,B 0,C 180,E1 35660.472,E2 35660.472} C_VEL
LIN {X 0,Y 751.879,Z 310.565,A -85,B 0,C 180,E1 35658.131,E2 35658.131} C_VEL
LIN {X 0,Y 751.887,Z 310.564,A -85,B 0,C 180,E1 35655.82,E2 35655.82} C_VEL
LIN {X 0,Y 751.972,Z 310.566,A -85,B 0,C 180,E1 35653.065,E2 35653.065} C_VEL
LIN {X 0,Y 751.903,Z 310.561,A -85,B 0,C 180,E1 35650.254,E2 35650.254} C_VEL
LIN {X 0,Y 751.89,Z 310.561,A -85,B 0,C 180,E1 35647.873,E2 35647.873} C_VEL
LIN {X 0,Y 751.903,Z 310.564,A -85,B 0,C 180,E1 35645.494,E2 35645.494} C_VEL
LIN {X 0,Y 751.979,Z 310.559,A -85,B 0,C 180,E1 35642.667,E2 35642.667} C_VEL
LIN {X 0,Y 751.906,Z 310.561,A -85,B 0,C 180,E1 35639.924,E2 35639.924} C_VEL
LIN {X 0,Y 751.903,Z 310.562,A -85,B 0,C 180,E1 35637.485,E2 35637.485} C_VEL
LIN {X 0,Y 751.966,Z 310.565,A -85,B 0,C 180,E1 35634.812,E2 35634.812} C_VEL
LIN {X 0,Y 751.926,Z 310.557,A -85,B 0,C 180,E1 35631.897,E2 35631.897} C_VEL
LIN {X 0,Y 751.911,Z 310.561,A -85,B 0,C 180,E1 35629.323,E2 35629.323} C_VEL
LIN {X 0,Y 751.975,Z 310.565,A -85,B 0,C 180,E1 35626.622,E2 35626.622} C_VEL
LIN {X 0,Y 751.934,Z 310.557,A -85,B 0,C 180,E1 35623.705,E2 35623.705} C_VEL
LIN {X 0,Y 751.919,Z 310.562,A -85,B 0,C 180,E1 35621.067,E2 35621.067} C_VEL
LIN {X 0,Y 751.973,Z 310.563,A -85,B 0,C 180,E1 35618.306,E2 35618.306} C_VEL
LIN {X 0,Y 751.935,Z 310.556,A -85,B 0,C 180,E1 35615.439,E2 35615.439} C_VEL
LIN {X 0,Y 751.94,Z 310.563,A -85,B 0,C 180,E1 35612.693,E2 35612.693} C_VEL
LIN {X 0,Y 751.976,Z 310.554,A -85,B 0,C 180,E1 35609.738,E2 35609.738} C_VEL
LIN {X 0,Y 751.929,Z 310.559,A -85,B 0,C 180,E1 35606.961,E2 35606.961} C_VEL
LIN {X 0,Y 751.974,Z 310.566,A -85,B 0,C 180,E1 35604.192,E2 35604.192} C_VEL
LIN {X 0,Y 751.952,Z 310.556,A -85,B 0,C 180,E1 35601.187,E2 35601.187} C_VEL
LIN {X 0,Y 751.955,Z 310.566,A -85,B 0,C 180,E1 35598.328,E2 35598.328} C_VEL
LIN {X 0,Y 751.975,Z 310.557,A -85,B 0,C 180,E1 35595.299,E2 35595.299} C_VEL
LIN {X 0,Y 751.996,Z 310.736,A -85,B 0,C 180,E1 35594.044,E2 35594.044} C_VEL
LIN {X 0,Y 753.405,Z 314.79,A -85,B 0,C 180,E1 35593.672,E2 35593.672} C_VEL
LIN {X 0,Y 753.396,Z 351.09,A -85,B 0,C 180,E1 35591.343,E2 35591.343} C_VEL
LIN {X 0,Y 753.838,Z 354.036,A -85,B 0,C 180,E1 35591.277,E2 35591.277} C_VEL
LIN {X 0,Y 753.62,Z 569.072,A -85,B 0,C 180,E1 35588.671,E2 35588.671} C_VEL
LIN {X 0,Y 753.408,Z 794.027,A -85,B 0,C 180,E1 35586.041,E2 35586.041} C_VEL
LIN {X 0,Y 753.35,Z 832.772,A -85,B 0,C 180,E1 35585.562,E2 35585.562} C_VEL
LIN {X 0,Y 753.27,Z 858.982,A -85,B 0,C 180,E1 35585.09,E2 35585.09} C_VEL
LIN {X 0,Y 753.186,Z 885.366,A -85,B 0,C 180,E1 35584.463,E2 35584.463} C_VEL
LIN {X 0,Y 753.086,Z 912.753,A -85,B 0,C 180,E1 35583.645,E2 35583.645} C_VEL
LIN {X 0,Y 752.952,Z 938.367,A -85,B 0,C 180,E1 35582.715,E2 35582.715} C_VEL
LIN {X 0,Y 752.856,Z 958.703,A -85,B 0,C 180,E1 35581.865,E2 35581.865} C_VEL
LIN {X 0,Y 752.76,Z 977.638,A -85,B 0,C 180,E1 35580.977,E2 35580.977} C_VEL
LIN {X 0,Y 752.664,Z 997.035,A -85,B 0,C 180,E1 35579.966,E2 35579.966} C_VEL
LIN {X 0,Y 752.556,Z 1018.075,A -85,B 0,C 180,E1 35578.748,E2 35578.748} C_VEL
LIN {X 0,Y 752.411,Z 1041.012,A -85,B 0,C 180,E1 35577.246,E2 35577.246} C_VEL
LIN {X 0,Y 752.345,Z 1059.059,A -85,B 0,C 180,E1 35575.928,E2 35575.928} C_VEL
LIN {X 0,Y 752.252,Z 1077.885,A -85,B 0,C 180,E1 35574.416,E2 35574.416} C_VEL
LIN {X 0,Y 752.168,Z 1096.907,A -85,B 0,C 180,E1 35572.695,E2 35572.695} C_VEL
LIN {X 0,Y 752.092,Z 1111.836,A -85,B 0,C 180,E1 35571.199,E2 35571.199} C_VEL
LIN {X 0,Y 752.069,Z 1126.513,A -85,B 0,C 180,E1 35569.574,E2 35569.574} C_VEL
LIN {X 0,Y 752.007,Z 1142.503,A -85,B 0,C 180,E1 35567.567,E2 35567.567} C_VEL
LIN {X 0,Y 751.954,Z 1153.718,A -85,B 0,C 180,E1 35565.972,E2 35565.972} C_VEL
LIN {X 0,Y 751.955,Z 1163.592,A -85,B 0,C 180,E1 35564.398,E2 35564.398} C_VEL
LIN {X 0,Y 751.942,Z 1172.291,A -85,B 0,C 180,E1 35562.83,E2 35562.83} C_VEL
LIN {X 0,Y 751.916,Z 1180.573,A -85,B 0,C 180,E1 35561.117,E2 35561.117} C_VEL
LIN {X 0,Y 751.92,Z 1188.481,A -85,B 0,C 180,E1 35559.182,E2 35559.182} C_VEL
LIN {X 0,Y 751.915,Z 1195.351,A -85,B 0,C 180,E1 35557.027,E2 35557.027} C_VEL
LIN {X 0,Y 751.918,Z 1200.041,A -85,B 0,C 180,E1 35555.035,E2 35555.035} C_VEL
LIN {X 0,Y 751.918,Z 1203.3,A -85,B 0,C 180,E1 35552.95,E2 35552.95} C_VEL
LIN {X 0,Y 751.914,Z 1204.715,A -85,B 0,C 180,E1 35550.991,E2 35550.991} C_VEL
LIN {X 0,Y 751.891,Z 1204.827,A -85,B 0,C 180,E1 35549.39,E2 35549.39} C_VEL
LIN {X 0,Y 751.906,Z 1203.828,A -85,B 0,C 180,E1 35547.561,E2 35547.561} C_VEL
LIN {X 0,Y 751.906,Z 1200.928,A -85,B 0,C 180,E1 35545.424,E2 35545.424} C_VEL
LIN {X 0,Y 751.909,Z 1196.371,A -85,B 0,C 180,E1 35543.357,E2 35543.357} C_VEL
LIN {X 0,Y 751.92,Z 1190.361,A -85,B 0,C 180,E1 35541.358,E2 35541.358} C_VEL
LIN {X 0,Y 751.905,Z 1182.355,A -85,B 0,C 180,E1 35539.271,E2 35539.271} C_VEL
LIN {X 0,Y 751.935,Z 1173.112,A -85,B 0,C 180,E1 35537.326,E2 35537.326} C_VEL
LIN {X 0,Y 751.955,Z 1164.058,A -85,B 0,C 180,E1 35535.681,E2 35535.681} C_VEL
LIN {X 0,Y 751.954,Z 1154.214,A -85,B 0,C 180,E1 35534.103,E2 35534.103} C_VEL
LIN {X 0,Y 752.006,Z 1143.086,A -85,B 0,C 180,E1 35532.513,E2 35532.513} C_VEL
LIN {X 0,Y 752.065,Z 1127.932,A -85,B 0,C 180,E1 35530.587,E2 35530.587} C_VEL
LIN {X 0,Y 752.088,Z 1112.616,A -85,B 0,C 180,E1 35528.883,E2 35528.883} C_VEL
LIN {X 0,Y 752.166,Z 1097.976,A -85,B 0,C 180,E1 35527.408,E2 35527.408} C_VEL
LIN {X 0,Y 752.232,Z 1079.859,A -85,B 0,C 180,E1 35525.75,E2 35525.75} C_VEL
LIN {X 0,Y 752.347,Z 1060.167,A -85,B 0,C 180,E1 35524.157,E2 35524.157} C_VEL
LIN {X 0,Y 752.409,Z 1042.84,A -85,B 0,C 180,E1 35522.883,E2 35522.883} C_VEL
LIN {X 0,Y 752.521,Z 1022.27,A -85,B 0,C 180,E1 35521.511,E2 35521.511} C_VEL
LIN {X 0,Y 752.657,Z 998.639,A -85,B 0,C 180,E1 35520.122,E2 35520.122} C_VEL
LIN {X 0,Y 752.754,Z 979.254,A -85,B 0,C 180,E1 35519.103,E2 35519.103} C_VEL
LIN {X 0,Y 752.85,Z 960.434,A -85,B 0,C 180,E1 35518.213,E2 35518.213} C_VEL
LIN {X 0,Y 752.948,Z 940.603,A -85,B 0,C 180,E1 35517.375,E2 35517.375} C_VEL
LIN {X 0,Y 753.037,Z 920.043,A -85,B 0,C 180,E1 35516.609,E2 35516.609} C_VEL
LIN {X 0,Y 753.158,Z 894.913,A -85,B 0,C 180,E1 35515.802,E2 35515.802} C_VEL
LIN {X 0,Y 753.243,Z 867.449,A -85,B 0,C 180,E1 35515.094,E2 35515.094} C_VEL
LIN {X 0,Y 753.331,Z 841.93,A -85,B 0,C 180,E1 35514.586,E2 35514.586} C_VEL
LIN {X 0,Y 753.38,Z 814.811,A -85,B 0,C 180,E1 35514.197,E2 35514.197} C_VEL
LIN {X 0,Y 753.595,Z 589.429,A -85,B 0,C 180,E1 35511.57,E2 35511.57} C_VEL
LIN {X 0,Y 753.804,Z 381.974,A -85,B 0,C 180,E1 35509.067,E2 35509.067} C_VEL
LIN {X 0,Y 753.652,Z 352.103,A -85,B 0,C 180,E1 35508.687,E2 35508.687} C_VEL
LIN {X 0,Y 753.275,Z 350.268,A -85,B 0,C 180,E1 35508.623,E2 35508.623} C_VEL
LIN {X 0,Y 753.328,Z 314.137,A -85,B 0,C 180,E1 35506.279,E2 35506.279} C_VEL
LIN {X 0,Y 751.972,Z 310.567,A -85,B 0,C 180,E1 35505.941,E2 35505.941} C_VEL
LIN {X 0,Y 751.942,Z 310.559,A -85,B 0,C 180,E1 35503.113,E2 35503.113} C_VEL
LIN {X 0,Y 751.966,Z 310.555,A -85,B 0,C 180,E1 35500.359,E2 35500.359} C_VEL
LIN {X 0,Y 751.947,Z 310.563,A -85,B 0,C 180,E1 35497.519,E2 35497.519} C_VEL
LIN {X 0,Y 751.952,Z 310.555,A -85,B 0,C 180,E1 35494.689,E2 35494.689} C_VEL
LIN {X 0,Y 751.97,Z 310.567,A -85,B 0,C 180,E1 35491.682,E2 35491.682} C_VEL
LIN {X 0,Y 751.927,Z 310.559,A -85,B 0,C 180,E1 35488.95,E2 35488.95} C_VEL
LIN {X 0,Y 751.974,Z 310.555,A -85,B 0,C 180,E1 35486.168,E2 35486.168} C_VEL
LIN {X 0,Y 751.943,Z 310.564,A -85,B 0,C 180,E1 35483.246,E2 35483.246} C_VEL
LIN {X 0,Y 751.927,Z 310.556,A -85,B 0,C 180,E1 35480.552,E2 35480.552} C_VEL
LIN {X 0,Y 751.971,Z 310.56,A -85,B 0,C 180,E1 35477.728,E2 35477.728} C_VEL
LIN {X 0,Y 751.926,Z 310.561,A -85,B 0,C 180,E1 35474.95,E2 35474.95} C_VEL
LIN {X 0,Y 751.92,Z 310.559,A -85,B 0,C 180,E1 35472.363,E2 35472.363} C_VEL
LIN {X 0,Y 751.974,Z 310.559,A -85,B 0,C 180,E1 35469.568,E2 35469.568} C_VEL
LIN {X 0,Y 751.917,Z 310.563,A -85,B 0,C 180,E1 35466.72,E2 35466.72} C_VEL
LIN {X 0,Y 751.911,Z 310.559,A -85,B 0,C 180,E1 35464.194,E2 35464.194} C_VEL
LIN {X 0,Y 751.977,Z 310.559,A -85,B 0,C 180,E1 35461.371,E2 35461.371} C_VEL
LIN {X 0,Y 751.911,Z 310.562,A -85,B 0,C 180,E1 35458.552,E2 35458.552} C_VEL
LIN {X 0,Y 751.9,Z 310.56,A -85,B 0,C 180,E1 35456.111,E2 35456.111} C_VEL
LIN {X 0,Y 751.904,Z 310.564,A -85,B 0,C 180,E1 35454.396,E2 35454.396} C_VEL
LIN {X 0,Y 750.886,Z 310.693,A -85,B 0,C 180,E1 35453.809,E2 35453.809} C_VEL
LIN {X 0,Y 744.473,Z 311.487,A -85,B 0,C 180,E1 35452.165,E2 35452.165} C_VEL
LIN {X 0,Y 743.973,Z 311.548,A -85,B 0,C 180,E1 35451.737,E2 35451.737} C_VEL
LIN {X 0,Y 744.012,Z 311.556,A -85,B 0,C 180,E1 35448.763,E2 35448.763} C_VEL
LIN {X 0,Y 743.955,Z 311.55,A -85,B 0,C 180,E1 35446.158,E2 35446.158} C_VEL
LIN {X 0,Y 743.951,Z 311.551,A -85,B 0,C 180,E1 35443.766,E2 35443.766} C_VEL
LIN {X 0,Y 744.017,Z 311.551,A -85,B 0,C 180,E1 35441.099,E2 35441.099} C_VEL
LIN {X 0,Y 743.964,Z 311.554,A -85,B 0,C 180,E1 35438.226,E2 35438.226} C_VEL
LIN {X 0,Y 743.94,Z 311.553,A -85,B 0,C 180,E1 35435.799,E2 35435.799} C_VEL
LIN {X 0,Y 743.941,Z 311.551,A -85,B 0,C 180,E1 35433.522,E2 35433.522} C_VEL
LIN {X 0,Y 743.987,Z 311.554,A -85,B 0,C 180,E1 35430.976,E2 35430.976} C_VEL
LIN {X 0,Y 743.954,Z 311.556,A -85,B 0,C 180,E1 35428,E2 35428} C_VEL
LIN {X 0,Y 743.93,Z 311.551,A -85,B 0,C 180,E1 35425.632,E2 35425.632} C_VEL
LIN {X 0,Y 743.927,Z 311.556,A -85,B 0,C 180,E1 35423.457,E2 35423.457} C_VEL
LIN {X 0,Y 743.93,Z 311.552,A -85,B 0,C 180,E1 35421.218,E2 35421.218} C_VEL
LIN {X 0,Y 744.007,Z 311.556,A -85,B 0,C 180,E1 35418.505,E2 35418.505} C_VEL
LIN {X 0,Y 743.942,Z 311.558,A -85,B 0,C 180,E1 35415.644,E2 35415.644} C_VEL
LIN {X 0,Y 743.93,Z 311.56,A -85,B 0,C 180,E1 35413.353,E2 35413.353} C_VEL
LIN {X 0,Y 744.006,Z 311.775,A -85,B 0,C 180,E1 35412.582,E2 35412.582} C_VEL
LIN {X 0,Y 746.481,Z 318.466,A -85,B 0,C 180,E1 35411.942,E2 35411.942} C_VEL
LIN {X 0,Y 746.611,Z 321.596,A -85,B 0,C 180,E1 35411.751,E2 35411.751} C_VEL
LIN {X 0,Y 747.727,Z 326.429,A -85,B 0,C 180,E1 35411.614,E2 35411.614} C_VEL
LIN {X 0,Y 747.416,Z 507.386,A -85,B 0,C 180,E1 35409.393,E2 35409.393} C_VEL
LIN {X 0,Y 746.99,Z 732.797,A -85,B 0,C 180,E1 35406.721,E2 35406.721} C_VEL
LIN {X 0,Y 746.822,Z 800.026,A -85,B 0,C 180,E1 35405.917,E2 35405.917} C_VEL
LIN {X 0,Y 746.676,Z 826.935,A -85,B 0,C 180,E1 35405.445,E2 35405.445} C_VEL
LIN {X 0,Y 746.507,Z 853.989,A -85,B 0,C 180,E1 35404.808,E2 35404.808} C_VEL
LIN {X 0,Y 746.313,Z 877.659,A -85,B 0,C 180,E1 35404.108,E2 35404.108} C_VEL
LIN {X 0,Y 746.123,Z 902.761,A -85,B 0,C 180,E1 35403.236,E2 35403.236} C_VEL
LIN {X 0,Y 745.825,Z 927.623,A -85,B 0,C 180,E1 35402.205,E2 35402.205} C_VEL
LIN {X 0,Y 745.631,Z 947.639,A -85,B 0,C 180,E1 35401.262,E2 35401.262} C_VEL
LIN {X 0,Y 745.438,Z 966.88,A -85,B 0,C 180,E1 35400.25,E2 35400.25} C_VEL
LIN {X 0,Y 745.234,Z 988.06,A -85,B 0,C 180,E1 35399.013,E2 35399.013} C_VEL
LIN {X 0,Y 744.949,Z 1011.325,A -85,B 0,C 180,E1 35397.474,E2 35397.474} C_VEL
LIN {X 0,Y 744.779,Z 1029.032,A -85,B 0,C 180,E1 35396.168,E2 35396.168} C_VEL
LIN {X 0,Y 744.62,Z 1048.108,A -85,B 0,C 180,E1 35394.62,E2 35394.62} C_VEL
LIN {X 0,Y 744.429,Z 1066.664,A -85,B 0,C 180,E1 35392.924,E2 35392.924} C_VEL
LIN {X 0,Y 744.313,Z 1081.571,A -85,B 0,C 180,E1 35391.415,E2 35391.415} C_VEL
LIN {X 0,Y 744.219,Z 1096.835,A -85,B 0,C 180,E1 35389.707,E2 35389.707} C_VEL
LIN {X 0,Y 744.092,Z 1112.181,A -85,B 0,C 180,E1 35387.76,E2 35387.76} C_VEL
LIN {X 0,Y 744.026,Z 1123.399,A -85,B 0,C 180,E1 35386.151,E2 35386.151} C_VEL
LIN {X 0,Y 744,Z 1133.331,A -85,B 0,C 180,E1 35384.555,E2 35384.555} C_VEL
LIN {X 0,Y 743.953,Z 1142.059,A -85,B 0,C 180,E1 35382.97,E2 35382.97} C_VEL
LIN {X 0,Y 743.946,Z 1149.654,A -85,B 0,C 180,E1 35381.395,E2 35381.395} C_VEL
LIN {X 0,Y 743.924,Z 1157.434,A -85,B 0,C 180,E1 35379.516,E2 35379.516} C_VEL
LIN {X 0,Y 743.914,Z 1164.126,A -85,B 0,C 180,E1 35377.491,E2 35377.491} C_VEL
LIN {X 0,Y 743.909,Z 1169.349,A -85,B 0,C 180,E1 35375.399,E2 35375.399} C_VEL
LIN {X 0,Y 743.91,Z 1172.831,A -85,B 0,C 180,E1 35373.313,E2 35373.313} C_VEL
LIN {X 0,Y 743.911,Z 1174.612,A -85,B 0,C 180,E1 35371.309,E2 35371.309} C_VEL
LIN {X 0,Y 743.889,Z 1174.862,A -85,B 0,C 180,E1 35369.461,E2 35369.461} C_VEL
LIN {X 0,Y 743.906,Z 1173.95,A -85,B 0,C 180,E1 35367.612,E2 35367.612} C_VEL
LIN {X 0,Y 743.906,Z 1171.127,A -85,B 0,C 180,E1 35365.452,E2 35365.452} C_VEL
LIN {X 0,Y 743.915,Z 1166.875,A -85,B 0,C 180,E1 35363.44,E2 35363.44} C_VEL
LIN {X 0,Y 743.929,Z 1161.047,A -85,B 0,C 180,E1 35361.42,E2 35361.42} C_VEL
LIN {X 0,Y 743.918,Z 1153.038,A -85,B 0,C 180,E1 35359.275,E2 35359.275} C_VEL
LIN {X 0,Y 743.971,Z 1143.347,A -85,B 0,C 180,E1 35357.188,E2 35357.188} C_VEL
LIN {X 0,Y 744.001,Z 1134.322,A -85,B 0,C 180,E1 35355.525,E2 35355.525} C_VEL
LIN {X 0,Y 744.023,Z 1124.473,A -85,B 0,C 180,E1 35353.923,E2 35353.923} C_VEL
LIN {X 0,Y 744.095,Z 1113.994,A -85,B 0,C 180,E1 35352.402,E2 35352.402} C_VEL
LIN {X 0,Y 744.174,Z 1100.933,A -85,B 0,C 180,E1 35350.7,E2 35350.7} C_VEL
LIN {X 0,Y 744.293,Z 1083.823,A -85,B 0,C 180,E1 35348.733,E2 35348.733} C_VEL
LIN {X 0,Y 744.418,Z 1069.291,A -85,B 0,C 180,E1 35347.243,E2 35347.243} C_VEL
LIN {X 0,Y 744.526,Z 1053.509,A -85,B 0,C 180,E1 35345.768,E2 35345.768} C_VEL
LIN {X 0,Y 744.776,Z 1032.41,A -85,B 0,C 180,E1 35344.003,E2 35344.003} C_VEL
LIN {X 0,Y 744.93,Z 1014.075,A -85,B 0,C 180,E1 35342.632,E2 35342.632} C_VEL
LIN {X 0,Y 745.119,Z 995.3,A -85,B 0,C 180,E1 35341.357,E2 35341.357} C_VEL
LIN {X 0,Y 745.409,Z 971.062,A -85,B 0,C 180,E1 35339.89,E2 35339.89} C_VEL
LIN {X 0,Y 745.616,Z 950.402,A -85,B 0,C 180,E1 35338.787,E2 35338.787} C_VEL
LIN {X 0,Y 745.808,Z 930.686,A -85,B 0,C 180,E1 35337.844,E2 35337.844} C_VEL
LIN {X 0,Y 746.002,Z 910.587,A -85,B 0,C 180,E1 35336.987,E2 35336.987} C_VEL
LIN {X 0,Y 746.189,Z 888.285,A -85,B 0,C 180,E1 35336.152,E2 35336.152} C_VEL
LIN {X 0,Y 746.457,Z 858.724,A -85,B 0,C 180,E1 35335.23,E2 35335.23} C_VEL
LIN {X 0,Y 746.651,Z 832.955,A -85,B 0,C 180,E1 35334.593,E2 35334.593} C_VEL
LIN {X 0,Y 746.806,Z 805.624,A -85,B 0,C 180,E1 35334.076,E2 35334.076} C_VEL
LIN {X 0,Y 746.909,Z 772.584,A -85,B 0,C 180,E1 35333.65,E2 35333.65} C_VEL
LIN {X 0,Y 747.35,Z 547.012,A -85,B 0,C 180,E1 35330.994,E2 35330.994} C_VEL
LIN {X 0,Y 747.713,Z 347.659,A -85,B 0,C 180,E1 35328.562,E2 35328.562} C_VEL
LIN {X 0,Y 747.574,Z 324.934,A -85,B 0,C 180,E1 35328.267,E2 35328.267} C_VEL
LIN {X 0,Y 746.47,Z 320.51,A -85,B 0,C 180,E1 35328.109,E2 35328.109} C_VEL
LIN {X 0,Y 746.394,Z 317.79,A -85,B 0,C 180,E1 35327.916,E2 35327.916} C_VEL
LIN {X 0,Y 743.974,Z 311.56,A -85,B 0,C 180,E1 35327.286,E2 35327.286} C_VEL
LIN {X 0,Y 743.94,Z 311.557,A -85,B 0,C 180,E1 35324.88,E2 35324.88} C_VEL
LIN {X 0,Y 743.933,Z 311.555,A -85,B 0,C 180,E1 35322.642,E2 35322.642} C_VEL
LIN {X 0,Y 743.935,Z 311.556,A -85,B 0,C 180,E1 35320.379,E2 35320.379} C_VEL
LIN {X 0,Y 743.991,Z 311.556,A -85,B 0,C 180,E1 35317.794,E2 35317.794} C_VEL
LIN {X 0,Y 743.949,Z 311.552,A -85,B 0,C 180,E1 35314.929,E2 35314.929} C_VEL
LIN {X 0,Y 743.926,Z 311.556,A -85,B 0,C 180,E1 35312.573,E2 35312.573} C_VEL
LIN {X 0,Y 743.925,Z 311.551,A -85,B 0,C 180,E1 35310.356,E2 35310.356} C_VEL
LIN {X 0,Y 743.931,Z 311.556,A -85,B 0,C 180,E1 35308.149,E2 35308.149} C_VEL
LIN {X 0,Y 743.98,Z 311.553,A -85,B 0,C 180,E1 35305.608,E2 35305.608} C_VEL
LIN {X 0,Y 743.956,Z 311.554,A -85,B 0,C 180,E1 35302.606,E2 35302.606} C_VEL
LIN {X 0,Y 743.939,Z 311.549,A -85,B 0,C 180,E1 35300.263,E2 35300.263} C_VEL
LIN {X 0,Y 743.941,Z 311.554,A -85,B 0,C 180,E1 35298.007,E2 35298.007} C_VEL
LIN {X 0,Y 743.965,Z 311.553,A -85,B 0,C 180,E1 35295.593,E2 35295.593} C_VEL
LIN {X 0,Y 743.992,Z 311.551,A -85,B 0,C 180,E1 35292.575,E2 35292.575} C_VEL
LIN {X 0,Y 743.952,Z 311.55,A -85,B 0,C 180,E1 35290.063,E2 35290.063} C_VEL
LIN {X 0,Y 743.953,Z 311.55,A -85,B 0,C 180,E1 35287.724,E2 35287.724} C_VEL
LIN {X 0,Y 744.013,Z 311.555,A -85,B 0,C 180,E1 35285.089,E2 35285.089} C_VEL
LIN {X 0,Y 743.98,Z 311.547,A -85,B 0,C 180,E1 35282.157,E2 35282.157} C_VEL
LIN {X 0,Y 743.96,Z 311.552,A -85,B 0,C 180,E1 35279.692,E2 35279.692} C_VEL
LIN {X 0,Y 743.988,Z 311.552,A -85,B 0,C 180,E1 35277.15,E2 35277.15} C_VEL
LIN {X 0,Y 743.999,Z 311.548,A -85,B 0,C 180,E1 35274.06,E2 35274.06} C_VEL
LIN {X 0,Y 743.968,Z 311.548,A -85,B 0,C 180,E1 35271.498,E2 35271.498} C_VEL
LIN {X 0,Y 744.011,Z 311.552,A -85,B 0,C 180,E1 35268.841,E2 35268.841} C_VEL
LIN {X 0,Y 744.002,Z 311.543,A -85,B 0,C 180,E1 35265.842,E2 35265.842} C_VEL
LIN {X 0,Y 743.977,Z 311.55,A -85,B 0,C 180,E1 35263.204,E2 35263.204} C_VEL
LIN {X 0,Y 744.037,Z 311.549,A -85,B 0,C 180,E1 35260.45,E2 35260.45} C_VEL
LIN {X 0,Y 743.993,Z 311.547,A -85,B 0,C 180,E1 35257.479,E2 35257.479} C_VEL
LIN {X 0,Y 743.999,Z 311.55,A -85,B 0,C 180,E1 35254.748,E2 35254.748} C_VEL
LIN {X 0,Y 744.039,Z 311.543,A -85,B 0,C 180,E1 35251.768,E2 35251.768} C_VEL
LIN {X 0,Y 743.989,Z 311.548,A -85,B 0,C 180,E1 35249.02,E2 35249.02} C_VEL
LIN {X 0,Y 744.037,Z 311.55,A -85,B 0,C 180,E1 35246.195,E2 35246.195} C_VEL
LIN {X 0,Y 744.011,Z 311.544,A -85,B 0,C 180,E1 35243.221,E2 35243.221} C_VEL
LIN {X 0,Y 744.02,Z 311.555,A -85,B 0,C 180,E1 35240.331,E2 35240.331} C_VEL
LIN {X 0,Y 744.029,Z 311.546,A -85,B 0,C 180,E1 35237.26,E2 35237.26} C_VEL
LIN {X 0,Y 744.015,Z 311.649,A -85,B 0,C 180,E1 35234.579,E2 35234.579} C_VEL
LIN {X 0,Y 745.358,Z 315.087,A -85,B 0,C 180,E1 35234.245,E2 35234.245} C_VEL
LIN {X 0,Y 746.918,Z 318.83,A -85,B 0,C 180,E1 35233.878,E2 35233.878} C_VEL
LIN {X 0,Y 746.794,Z 351.11,A -85,B 0,C 180,E1 35231.79,E2 35231.79} C_VEL
LIN {X 0,Y 747.807,Z 355.703,A -85,B 0,C 180,E1 35231.663,E2 35231.663} C_VEL
LIN {X 0,Y 747.36,Z 570.217,A -85,B 0,C 180,E1 35229.043,E2 35229.043} C_VEL
LIN {X 0,Y 746.927,Z 795.172,A -85,B 0,C 180,E1 35226.39,E2 35226.39} C_VEL
LIN {X 0,Y 746.816,Z 833.476,A -85,B 0,C 180,E1 35225.911,E2 35225.911} C_VEL
LIN {X 0,Y 746.657,Z 860.05,A -85,B 0,C 180,E1 35225.424,E2 35225.424} C_VEL
LIN {X 0,Y 746.485,Z 886.167,A -85,B 0,C 180,E1 35224.795,E2 35224.795} C_VEL
LIN {X 0,Y 746.271,Z 914.295,A -85,B 0,C 180,E1 35223.943,E2 35223.943} C_VEL
LIN {X 0,Y 746.006,Z 939.488,A -85,B 0,C 180,E1 35223.013,E2 35223.013} C_VEL
LIN {X 0,Y 745.813,Z 959.7,A -85,B 0,C 180,E1 35222.156,E2 35222.156} C_VEL
LIN {X 0,Y 745.618,Z 979.51,A -85,B 0,C 180,E1 35221.213,E2 35221.213} C_VEL
LIN {X 0,Y 745.411,Z 1001.051,A -85,B 0,C 180,E1 35220.066,E2 35220.066} C_VEL
LIN {X 0,Y 745.12,Z 1024.922,A -85,B 0,C 180,E1 35218.623,E2 35218.623} C_VEL
LIN {X 0,Y 744.926,Z 1043.447,A -85,B 0,C 180,E1 35217.368,E2 35217.368} C_VEL
LIN {X 0,Y 744.78,Z 1061.274,A -85,B 0,C 180,E1 35216.04,E2 35216.04} C_VEL
LIN {X 0,Y 744.532,Z 1083,A -85,B 0,C 180,E1 35214.233,E2 35214.233} C_VEL
LIN {X 0,Y 744.423,Z 1098.831,A -85,B 0,C 180,E1 35212.757,E2 35212.757} C_VEL
LIN {X 0,Y 744.289,Z 1114.958,A -85,B 0,C 180,E1 35211.102,E2 35211.102} C_VEL
LIN {X 0,Y 744.155,Z 1131.867,A -85,B 0,C 180,E1 35209.138,E2 35209.138} C_VEL
LIN {X 0,Y 744.097,Z 1144.252,A -85,B 0,C 180,E1 35207.517,E2 35207.517} C_VEL
LIN {X 0,Y 744.019,Z 1155.26,A -85,B 0,C 180,E1 35205.911,E2 35205.911} C_VEL
LIN {X 0,Y 744,Z 1165.921,A -85,B 0,C 180,E1 35204.157,E2 35204.157} C_VEL
LIN {X 0,Y 743.933,Z 1176.999,A -85,B 0,C 180,E1 35202.024,E2 35202.024} C_VEL
LIN {X 0,Y 743.93,Z 1185.541,A -85,B 0,C 180,E1 35200.062,E2 35200.062} C_VEL
LIN {X 0,Y 743.921,Z 1192.868,A -85,B 0,C 180,E1 35197.957,E2 35197.957} C_VEL
LIN {X 0,Y 743.911,Z 1198.261,A -85,B 0,C 180,E1 35195.936,E2 35195.936} C_VEL
LIN {X 0,Y 743.906,Z 1202.17,A -85,B 0,C 180,E1 35193.853,E2 35193.853} C_VEL
LIN {X 0,Y 743.906,Z 1204.381,A -85,B 0,C 180,E1 35191.771,E2 35191.771} C_VEL
LIN {X 0,Y 743.891,Z 1204.894,A -85,B 0,C 180,E1 35189.615,E2 35189.615} C_VEL
LIN {X 0,Y 743.908,Z 1203.979,A -85,B 0,C 180,E1 35187.689,E2 35187.689} C_VEL
LIN {X 0,Y 743.912,Z 1201.303,A -85,B 0,C 180,E1 35185.606,E2 35185.606} C_VEL
LIN {X 0,Y 743.919,Z 1197.153,A -85,B 0,C 180,E1 35183.595,E2 35183.595} C_VEL
LIN {X 0,Y 743.924,Z 1191.154,A -85,B 0,C 180,E1 35181.498,E2 35181.498} C_VEL
LIN {X 0,Y 743.919,Z 1183.319,A -85,B 0,C 180,E1 35179.389,E2 35179.389} C_VEL
LIN {X 0,Y 743.966,Z 1173.524,A -85,B 0,C 180,E1 35177.267,E2 35177.267} C_VEL
LIN {X 0,Y 743.999,Z 1164.525,A -85,B 0,C 180,E1 35175.604,E2 35175.604} C_VEL
LIN {X 0,Y 744.02,Z 1154.738,A -85,B 0,C 180,E1 35174.009,E2 35174.009} C_VEL
LIN {X 0,Y 744.097,Z 1144.252,A -85,B 0,C 180,E1 35172.483,E2 35172.483} C_VEL
LIN {X 0,Y 744.155,Z 1131.867,A -85,B 0,C 180,E1 35170.862,E2 35170.862} C_VEL
LIN {X 0,Y 744.287,Z 1114.958,A -85,B 0,C 180,E1 35168.898,E2 35168.898} C_VEL
LIN {X 0,Y 744.423,Z 1098.831,A -85,B 0,C 180,E1 35167.243,E2 35167.243} C_VEL
LIN {X 0,Y 744.541,Z 1082.148,A -85,B 0,C 180,E1 35165.691,E2 35165.691} C_VEL
LIN {X 0,Y 744.781,Z 1061.274,A -85,B 0,C 180,E1 35163.96,E2 35163.96} C_VEL
LIN {X 0,Y 744.926,Z 1043.446,A -85,B 0,C 180,E1 35162.632,E2 35162.632} C_VEL
LIN {X 0,Y 745.123,Z 1024.605,A -85,B 0,C 180,E1 35161.356,E2 35161.356} C_VEL
LIN {X 0,Y 745.415,Z 1000.247,A -85,B 0,C 180,E1 35159.89,E2 35159.89} C_VEL
LIN {X 0,Y 745.618,Z 979.51,A -85,B 0,C 180,E1 35158.787,E2 35158.787} C_VEL
LIN {X 0,Y 745.813,Z 959.701,A -85,B 0,C 180,E1 35157.844,E2 35157.844} C_VEL
LIN {X 0,Y 746.014,Z 938.371,A -85,B 0,C 180,E1 35156.942,E2 35156.942} C_VEL
LIN {X 0,Y 746.297,Z 911.449,A -85,B 0,C 180,E1 35155.966,E2 35155.966} C_VEL
LIN {X 0,Y 746.494,Z 885.167,A -85,B 0,C 180,E1 35155.178,E2 35155.178} C_VEL
LIN {X 0,Y 746.663,Z 858.731,A -85,B 0,C 180,E1 35154.548,E2 35154.548} C_VEL
LIN {X 0,Y 746.818,Z 832.089,A -85,B 0,C 180,E1 35154.068,E2 35154.068} C_VEL
LIN {X 0,Y 746.942,Z 789.255,A -85,B 0,C 180,E1 35153.541,E2 35153.541} C_VEL
LIN {X 0,Y 747.381,Z 562.103,A -85,B 0,C 180,E1 35150.86,E2 35150.86} C_VEL
LIN {X 0,Y 747.768,Z 354.754,A -85,B 0,C 180,E1 35148.323,E2 35148.323} C_VEL
LIN {X 0,Y 746.668,Z 350.268,A -85,B 0,C 180,E1 35148.174,E2 35148.174} C_VEL
LIN {X 0,Y 746.796,Z 318.367,A -85,B 0,C 180,E1 35146.082,E2 35146.082} C_VEL
LIN {X 0,Y 745.358,Z 315.087,A -85,B 0,C 180,E1 35145.755,E2 35145.755} C_VEL
LIN {X 0,Y 744.001,Z 311.555,A -85,B 0,C 180,E1 35145.383,E2 35145.383} C_VEL
LIN {X 0,Y 744.033,Z 311.547,A -85,B 0,C 180,E1 35142.573,E2 35142.573} C_VEL
LIN {X 0,Y 744.012,Z 311.554,A -85,B 0,C 180,E1 35139.57,E2 35139.57} C_VEL
LIN {X 0,Y 744.015,Z 311.544,A -85,B 0,C 180,E1 35136.73,E2 35136.73} C_VEL
LIN {X 0,Y 744.036,Z 311.55,A -85,B 0,C 180,E1 35133.712,E2 35133.712} C_VEL
LIN {X 0,Y 743.992,Z 311.547,A -85,B 0,C 180,E1 35130.89,E2 35130.89} C_VEL
LIN {X 0,Y 744.033,Z 311.544,A -85,B 0,C 180,E1 35128.145,E2 35128.145} C_VEL
LIN {X 0,Y 743.998,Z 311.55,A -85,B 0,C 180,E1 35125.216,E2 35125.216} C_VEL
LIN {X 0,Y 743.994,Z 311.547,A -85,B 0,C 180,E1 35122.521,E2 35122.521} C_VEL
LIN {X 0,Y 744.036,Z 311.548,A -85,B 0,C 180,E1 35119.606,E2 35119.606} C_VEL
LIN {X 0,Y 743.981,Z 311.55,A -85,B 0,C 180,E1 35116.795,E2 35116.795} C_VEL
LIN {X 0,Y 744.004,Z 311.542,A -85,B 0,C 180,E1 35114.158,E2 35114.158} C_VEL
LIN {X 0,Y 744.006,Z 311.552,A -85,B 0,C 180,E1 35111.08,E2 35111.08} C_VEL
LIN {X 0,Y 743.972,Z 311.547,A -85,B 0,C 180,E1 35108.424,E2 35108.424} C_VEL
LIN {X 0,Y 744.029,Z 311.546,A -85,B 0,C 180,E1 35105.707,E2 35105.707} C_VEL
LIN {X 0,Y 743.986,Z 311.551,A -85,B 0,C 180,E1 35102.773,E2 35102.773} C_VEL
LIN {X 0,Y 743.965,Z 311.551,A -85,B 0,C 180,E1 35100.231,E2 35100.231} C_VEL
LIN {X 0,Y 744.021,Z 311.545,A -85,B 0,C 180,E1 35097.535,E2 35097.535} C_VEL
LIN {X 0,Y 743.98,Z 311.554,A -85,B 0,C 180,E1 35094.602,E2 35094.602} C_VEL
LIN {X 0,Y 743.957,Z 311.549,A -85,B 0,C 180,E1 35092.098,E2 35092.098} C_VEL
LIN {X 0,Y 743.973,Z 311.548,A -85,B 0,C 180,E1 35091.737,E2 35091.737} C_VEL
LIN {X 0,Y 743.025,Z 311.675,A -85,B 0,C 180,E1 35091.144,E2 35091.144} C_VEL
LIN {X 0,Y 736.626,Z 312.465,A -85,B 0,C 180,E1 35089.483,E2 35089.483} C_VEL
LIN {X 0,Y 736.1,Z 312.538,A -85,B 0,C 180,E1 35089.052,E2 35089.052} C_VEL
LIN {X 0,Y 736.019,Z 312.539,A -85,B 0,C 180,E1 35086.24,E2 35086.24} C_VEL
LIN {X 0,Y 736.011,Z 312.539,A -85,B 0,C 180,E1 35083.829,E2 35083.829} C_VEL
LIN {X 0,Y 736.046,Z 312.541,A -85,B 0,C 180,E1 35081.301,E2 35081.301} C_VEL
LIN {X 0,Y 736.034,Z 312.544,A -85,B 0,C 180,E1 35078.306,E2 35078.306} C_VEL
LIN {X 0,Y 736.003,Z 312.542,A -85,B 0,C 180,E1 35075.863,E2 35075.863} C_VEL
LIN {X 0,Y 736.003,Z 312.54,A -85,B 0,C 180,E1 35073.54,E2 35073.54} C_VEL
LIN {X 0,Y 736.06,Z 312.543,A -85,B 0,C 180,E1 35070.901,E2 35070.901} C_VEL
LIN {X 0,Y 736.012,Z 312.545,A -85,B 0,C 180,E1 35067.961,E2 35067.961} C_VEL
LIN {X 0,Y 735.991,Z 312.539,A -85,B 0,C 180,E1 35065.586,E2 35065.586} C_VEL
LIN {X 0,Y 735.992,Z 312.546,A -85,B 0,C 180,E1 35063.276,E2 35063.276} C_VEL
LIN {X 0,Y 736.038,Z 312.54,A -85,B 0,C 180,E1 35060.724,E2 35060.724} C_VEL
LIN {X 0,Y 736.004,Z 312.546,A -85,B 0,C 180,E1 35057.741,E2 35057.741} C_VEL
LIN {X 0,Y 735.99,Z 312.548,A -85,B 0,C 180,E1 35055.382,E2 35055.382} C_VEL
LIN {X 0,Y 736.005,Z 312.643,A -85,B 0,C 180,E1 35053.095,E2 35053.095} C_VEL
LIN {X 0,Y 737.141,Z 315.759,A -85,B 0,C 180,E1 35052.791,E2 35052.791} C_VEL
LIN {X 0,Y 739.707,Z 321.445,A -85,B 0,C 180,E1 35052.233,E2 35052.233} C_VEL
LIN {X 0,Y 741.732,Z 327.817,A -85,B 0,C 180,E1 35052.009,E2 35052.009} C_VEL
LIN {X 0,Y 741.219,Z 509.98,A -85,B 0,C 180,E1 35049.756,E2 35049.756} C_VEL
LIN {X 0,Y 740.564,Z 735.364,A -85,B 0,C 180,E1 35047.063,E2 35047.063} C_VEL
LIN {X 0,Y 740.322,Z 800.307,A -85,B 0,C 180,E1 35046.279,E2 35046.279} C_VEL
LIN {X 0,Y 740.104,Z 827.46,A -85,B 0,C 180,E1 35045.797,E2 35045.797} C_VEL
LIN {X 0,Y 739.843,Z 854.204,A -85,B 0,C 180,E1 35045.162,E2 35045.162} C_VEL
LIN {X 0,Y 739.558,Z 877.851,A -85,B 0,C 180,E1 35044.458,E2 35044.458} C_VEL
LIN {X 0,Y 739.256,Z 903.083,A -85,B 0,C 180,E1 35043.573,E2 35043.573} C_VEL
LIN {X 0,Y 738.813,Z 928.148,A -85,B 0,C 180,E1 35042.525,E2 35042.525} C_VEL
LIN {X 0,Y 738.515,Z 948.544,A -85,B 0,C 180,E1 35041.552,E2 35041.552} C_VEL
LIN {X 0,Y 738.209,Z 969.447,A -85,B 0,C 180,E1 35040.435,E2 35040.435} C_VEL
LIN {X 0,Y 737.791,Z 994.25,A -85,B 0,C 180,E1 35038.934,E2 35038.934} C_VEL
LIN {X 0,Y 737.475,Z 1013.431,A -85,B 0,C 180,E1 35037.625,E2 35037.625} C_VEL
LIN {X 0,Y 737.223,Z 1031.089,A -85,B 0,C 180,E1 35036.296,E2 35036.296} C_VEL
LIN {X 0,Y 736.903,Z 1052.166,A -85,B 0,C 180,E1 35034.531,E2 35034.531} C_VEL
LIN {X 0,Y 736.691,Z 1068.378,A -85,B 0,C 180,E1 35033.009,E2 35033.009} C_VEL
LIN {X 0,Y 736.519,Z 1082.98,A -85,B 0,C 180,E1 35031.502,E2 35031.502} C_VEL
LIN {X 0,Y 736.346,Z 1099.584,A -85,B 0,C 180,E1 35029.596,E2 35029.596} C_VEL
LIN {X 0,Y 736.188,Z 1113.351,A -85,B 0,C 180,E1 35027.793,E2 35027.793} C_VEL
LIN {X 0,Y 736.097,Z 1123.927,A -85,B 0,C 180,E1 35026.249,E2 35026.249} C_VEL
LIN {X 0,Y 736.039,Z 1133.389,A -85,B 0,C 180,E1 35024.707,E2 35024.707} C_VEL
LIN {X 0,Y 735.982,Z 1142.3,A -85,B 0,C 180,E1 35023.067,E2 35023.067} C_VEL
LIN {X 0,Y 735.965,Z 1150.372,A -85,B 0,C 180,E1 35021.361,E2 35021.361} C_VEL
LIN {X 0,Y 735.938,Z 1158.316,A -85,B 0,C 180,E1 35019.383,E2 35019.383} C_VEL
LIN {X 0,Y 735.921,Z 1165.006,A -85,B 0,C 180,E1 35017.259,E2 35017.259} C_VEL
LIN {X 0,Y 735.911,Z 1169.808,A -85,B 0,C 180,E1 35015.223,E2 35015.223} C_VEL
LIN {X 0,Y 735.912,Z 1173.137,A -85,B 0,C 180,E1 35013.115,E2 35013.115} C_VEL
LIN {X 0,Y 735.91,Z 1174.679,A -85,B 0,C 180,E1 35011.09,E2 35011.09} C_VEL
LIN {X 0,Y 735.891,Z 1174.84,A -85,B 0,C 180,E1 35009.377,E2 35009.377} C_VEL
LIN {X 0,Y 735.905,Z 1173.873,A -85,B 0,C 180,E1 35007.508,E2 35007.508} C_VEL
LIN {X 0,Y 735.906,Z 1171.126,A -85,B 0,C 180,E1 35005.402,E2 35005.402} C_VEL
LIN {X 0,Y 735.913,Z 1166.765,A -85,B 0,C 180,E1 35003.325,E2 35003.325} C_VEL
LIN {X 0,Y 735.93,Z 1160.783,A -85,B 0,C 180,E1 35001.248,E2 35001.248} C_VEL
LIN {X 0,Y 735.934,Z 1152.863,A -85,B 0,C 180,E1 34999.114,E2 34999.114} C_VEL
LIN {X 0,Y 735.99,Z 1143.346,A -85,B 0,C 180,E1 34997.047,E2 34997.047} C_VEL
LIN {X 0,Y 736.039,Z 1134.321,A -85,B 0,C 180,E1 34995.365,E2 34995.365} C_VEL
LIN {X 0,Y 736.093,Z 1124.933,A -85,B 0,C 180,E1 34993.817,E2 34993.817} C_VEL
LIN {X 0,Y 736.189,Z 1114.574,A -85,B 0,C 180,E1 34992.288,E2 34992.288} C_VEL
LIN {X 0,Y 736.302,Z 1102.221,A -85,B 0,C 180,E1 34990.65,E2 34990.65} C_VEL
LIN {X 0,Y 736.487,Z 1086.152,A -85,B 0,C 180,E1 34988.747,E2 34988.747} C_VEL
LIN {X 0,Y 736.681,Z 1070.141,A -85,B 0,C 180,E1 34987.075,E2 34987.075} C_VEL
LIN {X 0,Y 736.853,Z 1054.373,A -85,B 0,C 180,E1 34985.579,E2 34985.579} C_VEL
LIN {X 0,Y 737.21,Z 1034.522,A -85,B 0,C 180,E1 34983.882,E2 34983.882} C_VEL
LIN {X 0,Y 737.462,Z 1014.673,A -85,B 0,C 180,E1 34982.375,E2 34982.375} C_VEL
LIN {X 0,Y 737.74,Z 996.302,A -85,B 0,C 180,E1 34981.111,E2 34981.111} C_VEL
LIN {X 0,Y 738.171,Z 973.464,A -85,B 0,C 180,E1 34979.698,E2 34979.698} C_VEL
LIN {X 0,Y 738.501,Z 950.305,A -85,B 0,C 180,E1 34978.447,E2 34978.447} C_VEL
LIN {X 0,Y 738.796,Z 930.154,A -85,B 0,C 180,E1 34977.477,E2 34977.477} C_VEL
LIN {X 0,Y 739.106,Z 908.451,A -85,B 0,C 180,E1 34976.551,E2 34976.551} C_VEL
LIN {X 0,Y 739.535,Z 881.367,A -85,B 0,C 180,E1 34975.564,E2 34975.564} C_VEL
LIN {X 0,Y 739.829,Z 855.331,A -85,B 0,C 180,E1 34974.779,E2 34974.779} C_VEL
LIN {X 0,Y 740.088,Z 829.014,A -85,B 0,C 180,E1 34974.146,E2 34974.146} C_VEL
LIN {X 0,Y 740.316,Z 802.286,A -85,B 0,C 180,E1 34973.661,E2 34973.661} C_VEL
LIN {X 0,Y 740.497,Z 758.528,A -85,B 0,C 180,E1 34973.118,E2 34973.118} C_VEL
LIN {X 0,Y 741.16,Z 534.076,A -85,B 0,C 180,E1 34970.447,E2 34970.447} C_VEL
LIN {X 0,Y 741.719,Z 336.348,A -85,B 0,C 180,E1 34968.009,E2 34968.009} C_VEL
LIN {X 0,Y 741.574,Z 327.176,A -85,B 0,C 180,E1 34967.881,E2 34967.881} C_VEL
LIN {X 0,Y 739.73,Z 321.457,A -85,B 0,C 180,E1 34967.679,E2 34967.679} C_VEL
LIN {X 0,Y 736.869,Z 315.279,A -85,B 0,C 180,E1 34967.066,E2 34967.066} C_VEL
LIN {X 0,Y 736.001,Z 312.55,A -85,B 0,C 180,E1 34966.789,E2 34966.789} C_VEL
LIN {X 0,Y 736.002,Z 312.547,A -85,B 0,C 180,E1 34964.503,E2 34964.503} C_VEL
LIN {X 0,Y 736.065,Z 312.544,A -85,B 0,C 180,E1 34961.835,E2 34961.835} C_VEL
LIN {X 0,Y 736.011,Z 312.546,A -85,B 0,C 180,E1 34958.976,E2 34958.976} C_VEL
LIN {X 0,Y 735.989,Z 312.546,A -85,B 0,C 180,E1 34956.594,E2 34956.594} C_VEL
LIN {X 0,Y 735.986,Z 312.539,A -85,B 0,C 180,E1 34954.312,E2 34954.312} C_VEL
LIN {X 0,Y 736.025,Z 312.546,A -85,B 0,C 180,E1 34951.81,E2 34951.81} C_VEL
LIN {X 0,Y 736.017,Z 312.544,A -85,B 0,C 180,E1 34948.811,E2 34948.811} C_VEL
LIN {X 0,Y 735.993,Z 312.541,A -85,B 0,C 180,E1 34946.375,E2 34946.375} C_VEL
LIN {X 0,Y 735.996,Z 312.542,A -85,B 0,C 180,E1 34944.089,E2 34944.089} C_VEL
LIN {X 0,Y 736.034,Z 312.544,A -85,B 0,C 180,E1 34941.602,E2 34941.602} C_VEL
LIN {X 0,Y 736.024,Z 312.542,A -85,B 0,C 180,E1 34938.535,E2 34938.535} C_VEL
LIN {X 0,Y 736.005,Z 312.541,A -85,B 0,C 180,E1 34936.09,E2 34936.09} C_VEL
LIN {X 0,Y 736.012,Z 312.538,A -85,B 0,C 180,E1 34933.753,E2 34933.753} C_VEL
LIN {X 0,Y 736.099,Z 312.54,A -85,B 0,C 180,E1 34930.963,E2 34930.963} C_VEL
LIN {X 0,Y 736.021,Z 312.536,A -85,B 0,C 180,E1 34928.122,E2 34928.122} C_VEL
LIN {X 0,Y 736.017,Z 312.542,A -85,B 0,C 180,E1 34925.692,E2 34925.692} C_VEL
LIN {X 0,Y 736.076,Z 312.539,A -85,B 0,C 180,E1 34923.037,E2 34923.037} C_VEL
LIN {X 0,Y 736.041,Z 312.539,A -85,B 0,C 180,E1 34920.078,E2 34920.078} C_VEL
LIN {X 0,Y 736.024,Z 312.538,A -85,B 0,C 180,E1 34917.586,E2 34917.586} C_VEL
LIN {X 0,Y 736.072,Z 312.539,A -85,B 0,C 180,E1 34914.934,E2 34914.934} C_VEL
LIN {X 0,Y 736.055,Z 312.533,A -85,B 0,C 180,E1 34911.957,E2 34911.957} C_VEL
LIN {X 0,Y 736.032,Z 312.537,A -85,B 0,C 180,E1 34909.353,E2 34909.353} C_VEL
LIN {X 0,Y 736.099,Z 312.539,A -85,B 0,C 180,E1 34906.569,E2 34906.569} C_VEL
LIN {X 0,Y 736.053,Z 312.535,A -85,B 0,C 180,E1 34903.668,E2 34903.668} C_VEL
LIN {X 0,Y 736.048,Z 312.541,A -85,B 0,C 180,E1 34900.972,E2 34900.972} C_VEL
LIN {X 0,Y 736.096,Z 312.537,A -85,B 0,C 180,E1 34898.065,E2 34898.065} C_VEL
LIN {X 0,Y 736.048,Z 312.534,A -85,B 0,C 180,E1 34895.266,E2 34895.266} C_VEL
LIN {X 0,Y 736.085,Z 312.543,A -85,B 0,C 180,E1 34892.493,E2 34892.493} C_VEL
LIN {X 0,Y 736.076,Z 312.532,A -85,B 0,C 180,E1 34889.451,E2 34889.451} C_VEL
LIN {X 0,Y 736.063,Z 312.541,A -85,B 0,C 180,E1 34886.621,E2 34886.621} C_VEL
LIN {X 0,Y 736.092,Z 312.533,A -85,B 0,C 180,E1 34883.657,E2 34883.657} C_VEL
LIN {X 0,Y 736.057,Z 312.539,A -85,B 0,C 180,E1 34880.826,E2 34880.826} C_VEL
LIN {X 0,Y 736.095,Z 312.544,A -85,B 0,C 180,E1 34877.988,E2 34877.988} C_VEL
LIN {X 0,Y 736.1,Z 312.632,A -85,B 0,C 180,E1 34875.122,E2 34875.122} C_VEL
LIN {X 0,Y 737.212,Z 315.778,A -85,B 0,C 180,E1 34874.818,E2 34874.818} C_VEL
LIN {X 0,Y 740.442,Z 322.825,A -85,B 0,C 180,E1 34874.09,E2 34874.09} C_VEL
LIN {X 0,Y 740.212,Z 351.071,A -85,B 0,C 180,E1 34872.247,E2 34872.247} C_VEL
LIN {X 0,Y 741.809,Z 357.782,A -85,B 0,C 180,E1 34872.049,E2 34872.049} C_VEL
LIN {X 0,Y 741.13,Z 571.489,A -85,B 0,C 180,E1 34869.419,E2 34869.419} C_VEL
LIN {X 0,Y 740.475,Z 796.023,A -85,B 0,C 180,E1 34866.749,E2 34866.749} C_VEL
LIN {X 0,Y 740.312,Z 833.872,A -85,B 0,C 180,E1 34866.271,E2 34866.271} C_VEL
LIN {X 0,Y 740.072,Z 860.594,A -85,B 0,C 180,E1 34865.776,E2 34865.776} C_VEL
LIN {X 0,Y 739.815,Z 886.57,A -85,B 0,C 180,E1 34865.143,E2 34865.143} C_VEL
LIN {X 0,Y 739.48,Z 914.932,A -85,B 0,C 180,E1 34864.274,E2 34864.274} C_VEL
LIN {X 0,Y 739.092,Z 939.492,A -85,B 0,C 180,E1 34863.361,E2 34863.361} C_VEL
LIN {X 0,Y 738.79,Z 960.697,A -85,B 0,C 180,E1 34862.453,E2 34862.453} C_VEL
LIN {X 0,Y 738.49,Z 981.244,A -85,B 0,C 180,E1 34861.46,E2 34861.46} C_VEL
LIN {X 0,Y 738.11,Z 1005.697,A -85,B 0,C 180,E1 34860.125,E2 34860.125} C_VEL
LIN {X 0,Y 737.732,Z 1026.91,A -85,B 0,C 180,E1 34858.804,E2 34858.804} C_VEL
LIN {X 0,Y 737.448,Z 1045.34,A -85,B 0,C 180,E1 34857.532,E2 34857.532} C_VEL
LIN {X 0,Y 737.182,Z 1066.231,A -85,B 0,C 180,E1 34855.937,E2 34855.937} C_VEL
LIN {X 0,Y 736.85,Z 1085.147,A -85,B 0,C 180,E1 34854.305,E2 34854.305} C_VEL
LIN {X 0,Y 736.68,Z 1100.568,A -85,B 0,C 180,E1 34852.838,E2 34852.838} C_VEL
LIN {X 0,Y 736.469,Z 1117.99,A -85,B 0,C 180,E1 34851.003,E2 34851.003} C_VEL
LIN {X 0,Y 736.294,Z 1132.514,A -85,B 0,C 180,E1 34849.268,E2 34849.268} C_VEL
LIN {X 0,Y 736.197,Z 1144.254,A -85,B 0,C 180,E1 34847.711,E2 34847.711} C_VEL
LIN {X 0,Y 736.09,Z 1154.739,A -85,B 0,C 180,E1 34846.168,E2 34846.168} C_VEL
LIN {X 0,Y 736.045,Z 1164.526,A -85,B 0,C 180,E1 34844.555,E2 34844.555} C_VEL
LIN {X 0,Y 735.988,Z 1174.756,A -85,B 0,C 180,E1 34842.634,E2 34842.634} C_VEL
LIN {X 0,Y 735.948,Z 1184.913,A -85,B 0,C 180,E1 34840.331,E2 34840.331} C_VEL
LIN {X 0,Y 735.928,Z 1192.136,A -85,B 0,C 180,E1 34838.28,E2 34838.28} C_VEL
LIN {X 0,Y 735.918,Z 1197.735,A -85,B 0,C 180,E1 34836.24,E2 34836.24} C_VEL
LIN {X 0,Y 735.912,Z 1201.928,A -85,B 0,C 180,E1 34834.051,E2 34834.051} C_VEL
LIN {X 0,Y 735.912,Z 1204.213,A -85,B 0,C 180,E1 34832.024,E2 34832.024} C_VEL
LIN {X 0,Y 735.898,Z 1204.939,A -85,B 0,C 180,E1 34829.766,E2 34829.766} C_VEL
LIN {X 0,Y 735.908,Z 1203.976,A -85,B 0,C 180,E1 34827.664,E2 34827.664} C_VEL
LIN {X 0,Y 735.91,Z 1201.303,A -85,B 0,C 180,E1 34825.558,E2 34825.558} C_VEL
LIN {X 0,Y 735.92,Z 1197.152,A -85,B 0,C 180,E1 34823.525,E2 34823.525} C_VEL
LIN {X 0,Y 735.931,Z 1191.151,A -85,B 0,C 180,E1 34821.405,E2 34821.405} C_VEL
LIN {X 0,Y 735.931,Z 1183.319,A -85,B 0,C 180,E1 34819.273,E2 34819.273} C_VEL
LIN {X 0,Y 735.999,Z 1173.525,A -85,B 0,C 180,E1 34817.127,E2 34817.127} C_VEL
LIN {X 0,Y 736.045,Z 1164.526,A -85,B 0,C 180,E1 34815.445,E2 34815.445} C_VEL
LIN {X 0,Y 736.092,Z 1154.646,A -85,B 0,C 180,E1 34813.817,E2 34813.817} C_VEL
LIN {X 0,Y 736.198,Z 1143.672,A -85,B 0,C 180,E1 34812.207,E2 34812.207} C_VEL
LIN {X 0,Y 736.364,Z 1129.29,A -85,B 0,C 180,E1 34810.322,E2 34810.322} C_VEL
LIN {X 0,Y 736.522,Z 1112.62,A -85,B 0,C 180,E1 34808.414,E2 34808.414} C_VEL
LIN {X 0,Y 736.685,Z 1097.979,A -85,B 0,C 180,E1 34806.906,E2 34806.906} C_VEL
LIN {X 0,Y 736.985,Z 1079.52,A -85,B 0,C 180,E1 34805.184,E2 34805.184} C_VEL
LIN {X 0,Y 737.229,Z 1060.167,A -85,B 0,C 180,E1 34803.587,E2 34803.587} C_VEL
LIN {X 0,Y 737.478,Z 1042.501,A -85,B 0,C 180,E1 34802.263,E2 34802.263} C_VEL
LIN {X 0,Y 737.895,Z 1020.413,A -85,B 0,C 180,E1 34800.77,E2 34800.77} C_VEL
LIN {X 0,Y 738.221,Z 997.841,A -85,B 0,C 180,E1 34799.431,E2 34799.431} C_VEL
LIN {X 0,Y 738.518,Z 977.732,A -85,B 0,C 180,E1 34798.362,E2 34798.362} C_VEL
LIN {X 0,Y 738.84,Z 956.624,A -85,B 0,C 180,E1 34797.361,E2 34797.361} C_VEL
LIN {X 0,Y 739.293,Z 929.68,A -85,B 0,C 180,E1 34796.257,E2 34796.257} C_VEL
LIN {X 0,Y 739.567,Z 907.054,A -85,B 0,C 180,E1 34795.472,E2 34795.472} C_VEL
LIN {X 0,Y 739.849,Z 883.684,A -85,B 0,C 180,E1 34794.78,E2 34794.78} C_VEL
LIN {X 0,Y 740.113,Z 856.978,A -85,B 0,C 180,E1 34794.148,E2 34794.148} C_VEL
LIN {X 0,Y 740.323,Z 829.712,A -85,B 0,C 180,E1 34793.667,E2 34793.667} C_VEL
LIN {X 0,Y 740.656,Z 731.68,A -85,B 0,C 180,E1 34792.495,E2 34792.495} C_VEL
LIN {X 0,Y 741.332,Z 508.761,A -85,B 0,C 180,E1 34789.82,E2 34789.82} C_VEL
LIN {X 0,Y 741.697,Z 356.62,A -85,B 0,C 180,E1 34787.928,E2 34787.928} C_VEL
LIN {X 0,Y 740.099,Z 350.268,A -85,B 0,C 180,E1 34787.718,E2 34787.718} C_VEL
LIN {X 0,Y 740.315,Z 322.5,A -85,B 0,C 180,E1 34785.878,E2 34785.878} C_VEL
LIN {X 0,Y 737.212,Z 315.778,A -85,B 0,C 180,E1 34785.182,E2 34785.182} C_VEL
LIN {X 0,Y 736.091,Z 312.54,A -85,B 0,C 180,E1 34784.842,E2 34784.842} C_VEL
LIN {X 0,Y 736.085,Z 312.538,A -85,B 0,C 180,E1 34781.729,E2 34781.729} C_VEL
LIN {X 0,Y 736.071,Z 312.536,A -85,B 0,C 180,E1 34778.873,E2 34778.873} C_VEL
LIN {X 0,Y 736.091,Z 312.541,A -85,B 0,C 180,E1 34775.932,E2 34775.932} C_VEL
LIN {X 0,Y 736.053,Z 312.538,A -85,B 0,C 180,E1 34773.1,E2 34773.1} C_VEL
LIN {X 0,Y 736.098,Z 312.532,A -85,B 0,C 180,E1 34770.244,E2 34770.244} C_VEL
LIN {X 0,Y 736.068,Z 312.541,A -85,B 0,C 180,E1 34767.33,E2 34767.33} C_VEL
LIN {X 0,Y 736.058,Z 312.532,A -85,B 0,C 180,E1 34764.562,E2 34764.562} C_VEL
LIN {X 0,Y 736.096,Z 312.543,A -85,B 0,C 180,E1 34761.6,E2 34761.6} C_VEL
LIN {X 0,Y 736.044,Z 312.539,A -85,B 0,C 180,E1 34758.864,E2 34758.864} C_VEL
LIN {X 0,Y 736.07,Z 312.534,A -85,B 0,C 180,E1 34756.169,E2 34756.169} C_VEL
LIN {X 0,Y 736.067,Z 312.543,A -85,B 0,C 180,E1 34753.105,E2 34753.105} C_VEL
LIN {X 0,Y 736.037,Z 312.536,A -85,B 0,C 180,E1 34750.422,E2 34750.422} C_VEL
LIN {X 0,Y 736.097,Z 312.532,A -85,B 0,C 180,E1 34747.65,E2 34747.65} C_VEL
LIN {X 0,Y 736.043,Z 312.539,A -85,B 0,C 180,E1 34744.753,E2 34744.753} C_VEL
LIN {X 0,Y 736.031,Z 312.535,A -85,B 0,C 180,E1 34742.18,E2 34742.18} C_VEL
LIN {X 0,Y 736.098,Z 312.539,A -85,B 0,C 180,E1 34739.377,E2 34739.377} C_VEL
LIN {X 0,Y 736.031,Z 312.538,A -85,B 0,C 180,E1 34736.495,E2 34736.495} C_VEL
LIN {X 0,Y 736.023,Z 312.54,A -85,B 0,C 180,E1 34733.996,E2 34733.996} C_VEL
LIN {X 0,Y 736.096,Z 312.535,A -85,B 0,C 180,E1 34731.249,E2 34731.249} C_VEL
LIN {X 0,Y 736.1,Z 312.538,A -85,B 0,C 180,E1 34729.052,E2 34729.052} C_VEL
LIN {X 0,Y 735.121,Z 312.669,A -85,B 0,C 180,E1 34728.452,E2 34728.452} C_VEL
LIN {X 0,Y 728.653,Z 313.465,A -85,B 0,C 180,E1 34726.774,E2 34726.774} C_VEL
LIN {X 0,Y 728.087,Z 313.527,A -85,B 0,C 180,E1 34726.337,E2 34726.337} C_VEL
LIN {X 0,Y 728.072,Z 313.528,A -85,B 0,C 180,E1 34723.894,E2 34723.894} C_VEL
LIN {X 0,Y 728.093,Z 313.53,A -85,B 0,C 180,E1 34721.421,E2 34721.421} C_VEL
LIN {X 0,Y 728.097,Z 313.533,A -85,B 0,C 180,E1 34718.32,E2 34718.32} C_VEL
LIN {X 0,Y 728.064,Z 313.531,A -85,B 0,C 180,E1 34715.842,E2 34715.842} C_VEL
LIN {X 0,Y 728.066,Z 313.528,A -85,B 0,C 180,E1 34713.491,E2 34713.491} C_VEL
LIN {X 0,Y 728.159,Z 313.529,A -85,B 0,C 180,E1 34710.684,E2 34710.684} C_VEL
LIN {X 0,Y 728.067,Z 313.535,A -85,B 0,C 180,E1 34707.894,E2 34707.894} C_VEL
LIN {X 0,Y 728.052,Z 313.526,A -85,B 0,C 180,E1 34705.54,E2 34705.54} C_VEL
LIN {X 0,Y 728.058,Z 313.535,A -85,B 0,C 180,E1 34703.192,E2 34703.192} C_VEL
LIN {X 0,Y 728.146,Z 313.53,A -85,B 0,C 180,E1 34700.384,E2 34700.384} C_VEL
LIN {X 0,Y 728.055,Z 313.536,A -85,B 0,C 180,E1 34697.598,E2 34697.598} C_VEL
LIN {X 0,Y 728.05,Z 313.539,A -85,B 0,C 180,E1 34695.318,E2 34695.318} C_VEL
LIN {X 0,Y 728.09,Z 313.707,A -85,B 0,C 180,E1 34693.604,E2 34693.604} C_VEL
LIN {X 0,Y 729.495,Z 317.221,A -85,B 0,C 180,E1 34693.244,E2 34693.244} C_VEL
LIN {X 0,Y 731.509,Z 321.516,A -85,B 0,C 180,E1 34692.819,E2 34692.819} C_VEL
LIN {X 0,Y 735.022,Z 327.318,A -85,B 0,C 180,E1 34692.49,E2 34692.49} C_VEL
LIN {X 0,Y 735.767,Z 330.924,A -85,B 0,C 180,E1 34692.39,E2 34692.39} C_VEL
LIN {X 0,Y 735.035,Z 517.407,A -85,B 0,C 180,E1 34690.066,E2 34690.066} C_VEL
LIN {X 0,Y 734.145,Z 742.863,A -85,B 0,C 180,E1 34687.353,E2 34687.353} C_VEL
LIN {X 0,Y 733.85,Z 800.941,A -85,B 0,C 180,E1 34686.642,E2 34686.642} C_VEL
LIN {X 0,Y 733.556,Z 828.291,A -85,B 0,C 180,E1 34686.149,E2 34686.149} C_VEL
LIN {X 0,Y 733.207,Z 854.535,A -85,B 0,C 180,E1 34685.519,E2 34685.519} C_VEL
LIN {X 0,Y 732.825,Z 878.678,A -85,B 0,C 180,E1 34684.793,E2 34684.793} C_VEL
LIN {X 0,Y 732.397,Z 903.933,A -85,B 0,C 180,E1 34683.895,E2 34683.895} C_VEL
LIN {X 0,Y 731.859,Z 927.755,A -85,B 0,C 180,E1 34682.892,E2 34682.892} C_VEL
LIN {X 0,Y 731.432,Z 948.344,A -85,B 0,C 180,E1 34681.904,E2 34681.904} C_VEL
LIN {X 0,Y 731.014,Z 969.46,A -85,B 0,C 180,E1 34680.767,E2 34680.767} C_VEL
LIN {X 0,Y 730.48,Z 994.261,A -85,B 0,C 180,E1 34679.252,E2 34679.252} C_VEL
LIN {X 0,Y 730.041,Z 1013.44,A -85,B 0,C 180,E1 34677.93,E2 34677.93} C_VEL
LIN {X 0,Y 729.68,Z 1031.52,A -85,B 0,C 180,E1 34676.556,E2 34676.556} C_VEL
LIN {X 0,Y 729.256,Z 1053.104,A -85,B 0,C 180,E1 34674.719,E2 34674.719} C_VEL
LIN {X 0,Y 728.96,Z 1068.894,A -85,B 0,C 180,E1 34673.217,E2 34673.217} C_VEL
LIN {X 0,Y 728.726,Z 1084.546,A -85,B 0,C 180,E1 34671.575,E2 34671.575} C_VEL
LIN {X 0,Y 728.462,Z 1101.524,A -85,B 0,C 180,E1 34669.567,E2 34669.567} C_VEL
LIN {X 0,Y 728.288,Z 1113.939,A -85,B 0,C 180,E1 34667.91,E2 34667.91} C_VEL
LIN {X 0,Y 728.166,Z 1124.821,A -85,B 0,C 180,E1 34666.292,E2 34666.292} C_VEL
LIN {X 0,Y 728.09,Z 1134.736,A -85,B 0,C 180,E1 34664.636,E2 34664.636} C_VEL
LIN {X 0,Y 728.026,Z 1145.338,A -85,B 0,C 180,E1 34662.613,E2 34662.613} C_VEL
LIN {X 0,Y 727.961,Z 1155.053,A -85,B 0,C 180,E1 34660.366,E2 34660.366} C_VEL
LIN {X 0,Y 727.937,Z 1162.242,A -85,B 0,C 180,E1 34658.292,E2 34658.292} C_VEL
LIN {X 0,Y 727.924,Z 1167.809,A -85,B 0,C 180,E1 34656.23,E2 34656.23} C_VEL
LIN {X 0,Y 727.915,Z 1171.982,A -85,B 0,C 180,E1 34654.017,E2 34654.017} C_VEL
LIN {X 0,Y 727.912,Z 1174.237,A -85,B 0,C 180,E1 34651.968,E2 34651.968} C_VEL
LIN {X 0,Y 727.894,Z 1174.929,A -85,B 0,C 180,E1 34649.685,E2 34649.685} C_VEL
LIN {X 0,Y 727.907,Z 1174.012,A -85,B 0,C 180,E1 34647.638,E2 34647.638} C_VEL
LIN {X 0,Y 727.909,Z 1171.375,A -85,B 0,C 180,E1 34645.509,E2 34645.509} C_VEL
LIN {X 0,Y 727.92,Z 1167.264,A -85,B 0,C 180,E1 34643.454,E2 34643.454} C_VEL
LIN {X 0,Y 727.938,Z 1161.292,A -85,B 0,C 180,E1 34641.31,E2 34641.31} C_VEL
LIN {X 0,Y 727.944,Z 1153.818,A -85,B 0,C 180,E1 34639.234,E2 34639.234} C_VEL
LIN {X 0,Y 728.017,Z 1143.755,A -85,B 0,C 180,E1 34636.983,E2 34636.983} C_VEL
LIN {X 0,Y 728.08,Z 1134.317,A -85,B 0,C 180,E1 34635.201,E2 34635.201} C_VEL
LIN {X 0,Y 728.176,Z 1124.505,A -85,B 0,C 180,E1 34633.569,E2 34633.569} C_VEL
LIN {X 0,Y 728.298,Z 1113.408,A -85,B 0,C 180,E1 34631.925,E2 34631.925} C_VEL
LIN {X 0,Y 728.519,Z 1098.992,A -85,B 0,C 180,E1 34630.017,E2 34630.017} C_VEL
LIN {X 0,Y 728.747,Z 1083.036,A -85,B 0,C 180,E1 34628.172,E2 34628.172} C_VEL
LIN {X 0,Y 728.959,Z 1068.429,A -85,B 0,C 180,E1 34626.647,E2 34626.647} C_VEL
LIN {X 0,Y 729.302,Z 1051.744,A -85,B 0,C 180,E1 34625.066,E2 34625.066} C_VEL
LIN {X 0,Y 729.684,Z 1030.952,A -85,B 0,C 180,E1 34623.309,E2 34623.309} C_VEL
LIN {X 0,Y 730.06,Z 1012.851,A -85,B 0,C 180,E1 34621.937,E2 34621.937} C_VEL
LIN {X 0,Y 730.556,Z 992.083,A -85,B 0,C 180,E1 34620.514,E2 34620.514} C_VEL
LIN {X 0,Y 731.019,Z 968.638,A -85,B 0,C 180,E1 34619.097,E2 34619.097} C_VEL
LIN {X 0,Y 731.427,Z 948.515,A -85,B 0,C 180,E1 34618.014,E2 34618.014} C_VEL
LIN {X 0,Y 731.858,Z 927.826,A -85,B 0,C 180,E1 34617.021,E2 34617.021} C_VEL
LIN {X 0,Y 732.442,Z 902.543,A -85,B 0,C 180,E1 34615.96,E2 34615.96} C_VEL
LIN {X 0,Y 732.844,Z 876.986,A -85,B 0,C 180,E1 34615.063,E2 34615.063} C_VEL
LIN {X 0,Y 733.214,Z 853.819,A -85,B 0,C 180,E1 34614.372,E2 34614.372} C_VEL
LIN {X 0,Y 733.581,Z 827.226,A -85,B 0,C 180,E1 34613.739,E2 34613.739} C_VEL
LIN {X 0,Y 733.855,Z 799.882,A -85,B 0,C 180,E1 34613.252,E2 34613.252} C_VEL
LIN {X 0,Y 734.3,Z 701.697,A -85,B 0,C 180,E1 34612.069,E2 34612.069} C_VEL
LIN {X 0,Y 735.155,Z 486.766,A -85,B 0,C 180,E1 34609.468,E2 34609.468} C_VEL
LIN {X 0,Y 735.747,Z 329.908,A -85,B 0,C 180,E1 34607.506,E2 34607.506} C_VEL
LIN {X 0,Y 734.383,Z 325.865,A -85,B 0,C 180,E1 34607.356,E2 34607.356} C_VEL
LIN {X 0,Y 731.021,Z 320.79,A -85,B 0,C 180,E1 34607.036,E2 34607.036} C_VEL
LIN {X 0,Y 728.113,Z 313.775,A -85,B 0,C 180,E1 34606.312,E2 34606.312} C_VEL
LIN {X 0,Y 728.132,Z 313.535,A -85,B 0,C 180,E1 34603.87,E2 34603.87} C_VEL
LIN {X 0,Y 728.069,Z 313.536,A -85,B 0,C 180,E1 34600.947,E2 34600.947} C_VEL
LIN {X 0,Y 728.052,Z 313.535,A -85,B 0,C 180,E1 34598.609,E2 34598.609} C_VEL
LIN {X 0,Y 728.055,Z 313.535,A -85,B 0,C 180,E1 34596.279,E2 34596.279} C_VEL
LIN {X 0,Y 728.14,Z 313.527,A -85,B 0,C 180,E1 34593.507,E2 34593.507} C_VEL
LIN {X 0,Y 728.061,Z 313.526,A -85,B 0,C 180,E1 34590.718,E2 34590.718} C_VEL
LIN {X 0,Y 728.051,Z 313.534,A -85,B 0,C 180,E1 34588.372,E2 34588.372} C_VEL
LIN {X 0,Y 728.057,Z 313.53,A -85,B 0,C 180,E1 34586.071,E2 34586.071} C_VEL
LIN {X 0,Y 728.133,Z 313.532,A -85,B 0,C 180,E1 34583.382,E2 34583.382} C_VEL
LIN {X 0,Y 728.074,Z 313.523,A -85,B 0,C 180,E1 34580.5,E2 34580.5} C_VEL
LIN {X 0,Y 728.063,Z 313.532,A -85,B 0,C 180,E1 34578.082,E2 34578.082} C_VEL
LIN {X 0,Y 728.078,Z 313.53,A -85,B 0,C 180,E1 34575.697,E2 34575.697} C_VEL
LIN {X 0,Y 728.145,Z 313.529,A -85,B 0,C 180,E1 34572.773,E2 34572.773} C_VEL
LIN {X 0,Y 728.075,Z 313.527,A -85,B 0,C 180,E1 34570.045,E2 34570.045} C_VEL
LIN {X 0,Y 728.078,Z 313.526,A -85,B 0,C 180,E1 34567.655,E2 34567.655} C_VEL
LIN {X 0,Y 728.16,Z 313.529,A -85,B 0,C 180,E1 34564.884,E2 34564.884} C_VEL
LIN {X 0,Y 728.087,Z 313.524,A -85,B 0,C 180,E1 34561.968,E2 34561.968} C_VEL
LIN {X 0,Y 728.088,Z 313.531,A -85,B 0,C 180,E1 34559.449,E2 34559.449} C_VEL
LIN {X 0,Y 728.16,Z 313.522,A -85,B 0,C 180,E1 34556.615,E2 34556.615} C_VEL
LIN {X 0,Y 728.096,Z 313.528,A -85,B 0,C 180,E1 34553.772,E2 34553.772} C_VEL
LIN {X 0,Y 728.099,Z 313.526,A -85,B 0,C 180,E1 34551.232,E2 34551.232} C_VEL
LIN {X 0,Y 728.16,Z 313.527,A -85,B 0,C 180,E1 34548.354,E2 34548.354} C_VEL
LIN {X 0,Y 728.101,Z 313.521,A -85,B 0,C 180,E1 34545.526,E2 34545.526} C_VEL
LIN {X 0,Y 728.124,Z 313.53,A -85,B 0,C 180,E1 34542.828,E2 34542.828} C_VEL
LIN {X 0,Y 728.13,Z 313.517,A -85,B 0,C 180,E1 34539.699,E2 34539.699} C_VEL
LIN {X 0,Y 728.112,Z 313.53,A -85,B 0,C 180,E1 34536.934,E2 34536.934} C_VEL
LIN {X 0,Y 728.155,Z 313.526,A -85,B 0,C 180,E1 34534.08,E2 34534.08} C_VEL
LIN {X 0,Y 728.117,Z 313.524,A -85,B 0,C 180,E1 34531.273,E2 34531.273} C_VEL
LIN {X 0,Y 728.142,Z 313.531,A -85,B 0,C 180,E1 34528.453,E2 34528.453} C_VEL
LIN {X 0,Y 728.139,Z 313.522,A -85,B 0,C 180,E1 34525.338,E2 34525.338} C_VEL
LIN {X 0,Y 728.135,Z 313.526,A -85,B 0,C 180,E1 34522.431,E2 34522.431} C_VEL
LIN {X 0,Y 728.157,Z 313.525,A -85,B 0,C 180,E1 34519.391,E2 34519.391} C_VEL
LIN {X 0,Y 728.128,Z 313.534,A -85,B 0,C 180,E1 34516.472,E2 34516.472} C_VEL
LIN {X 0,Y 728.172,Z 313.713,A -85,B 0,C 180,E1 34515.675,E2 34515.675} C_VEL
LIN {X 0,Y 729.547,Z 317.134,A -85,B 0,C 180,E1 34515.324,E2 34515.324} C_VEL
LIN {X 0,Y 733.967,Z 326.802,A -85,B 0,C 180,E1 34514.308,E2 34514.308} C_VEL
LIN {X 0,Y 733.707,Z 351.152,A -85,B 0,C 180,E1 34512.709,E2 34512.709} C_VEL
LIN {X 0,Y 735.845,Z 360.005,A -85,B 0,C 180,E1 34512.441,E2 34512.441} C_VEL
LIN {X 0,Y 734.932,Z 573.194,A -85,B 0,C 180,E1 34509.796,E2 34509.796} C_VEL
LIN {X 0,Y 734.051,Z 797.462,A -85,B 0,C 180,E1 34507.107,E2 34507.107} C_VEL
LIN {X 0,Y 733.835,Z 834.527,A -85,B 0,C 180,E1 34506.632,E2 34506.632} C_VEL
LIN {X 0,Y 733.512,Z 861.684,A -85,B 0,C 180,E1 34506.122,E2 34506.122} C_VEL
LIN {X 0,Y 733.163,Z 887.558,A -85,B 0,C 180,E1 34505.482,E2 34505.482} C_VEL
LIN {X 0,Y 732.692,Z 916.215,A -85,B 0,C 180,E1 34504.589,E2 34504.589} C_VEL
LIN {X 0,Y 732.218,Z 939.494,A -85,B 0,C 180,E1 34503.716,E2 34503.716} C_VEL
LIN {X 0,Y 731.8,Z 960.601,A -85,B 0,C 180,E1 34502.807,E2 34502.807} C_VEL
LIN {X 0,Y 731.386,Z 982.098,A -85,B 0,C 180,E1 34501.757,E2 34501.757} C_VEL
LIN {X 0,Y 730.852,Z 1007.164,A -85,B 0,C 180,E1 34500.365,E2 34500.365} C_VEL
LIN {X 0,Y 730.377,Z 1027.574,A -85,B 0,C 180,E1 34499.077,E2 34499.077} C_VEL
LIN {X 0,Y 729.986,Z 1046.473,A -85,B 0,C 180,E1 34497.755,E2 34497.755} C_VEL
LIN {X 0,Y 729.556,Z 1068.744,A -85,B 0,C 180,E1 34496.012,E2 34496.012} C_VEL
LIN {X 0,Y 729.184,Z 1085.987,A -85,B 0,C 180,E1 34494.5,E2 34494.5} C_VEL
LIN {X 0,Y 728.938,Z 1102.248,A -85,B 0,C 180,E1 34492.927,E2 34492.927} C_VEL
LIN {X 0,Y 728.633,Z 1120.124,A -85,B 0,C 180,E1 34490.987,E2 34490.987} C_VEL
LIN {X 0,Y 728.422,Z 1133.805,A -85,B 0,C 180,E1 34489.318,E2 34489.318} C_VEL
LIN {X 0,Y 728.291,Z 1145.42,A -85,B 0,C 180,E1 34487.745,E2 34487.745} C_VEL
LIN {X 0,Y 728.151,Z 1156.94,A -85,B 0,C 180,E1 34486.005,E2 34486.005} C_VEL
LIN {X 0,Y 728.047,Z 1169.422,A -85,B 0,C 180,E1 34483.825,E2 34483.825} C_VEL
LIN {X 0,Y 727.972,Z 1178.074,A -85,B 0,C 180,E1 34482.05,E2 34482.05} C_VEL
LIN {X 0,Y 727.953,Z 1185.838,A -85,B 0,C 180,E1 34480.206,E2 34480.206} C_VEL
LIN {X 0,Y 727.927,Z 1193.111,A -85,B 0,C 180,E1 34478.054,E2 34478.054} C_VEL
LIN {X 0,Y 727.914,Z 1198.422,A -85,B 0,C 180,E1 34475.992,E2 34475.992} C_VEL
LIN {X 0,Y 727.907,Z 1202.278,A -85,B 0,C 180,E1 34473.859,E2 34473.859} C_VEL
LIN {X 0,Y 727.908,Z 1204.493,A -85,B 0,C 180,E1 34471.653,E2 34471.653} C_VEL
LIN {X 0,Y 727.89,Z 1204.872,A -85,B 0,C 180,E1 34469.528,E2 34469.528} C_VEL
LIN {X 0,Y 727.906,Z 1203.905,A -85,B 0,C 180,E1 34467.56,E2 34467.56} C_VEL
LIN {X 0,Y 727.907,Z 1201.178,A -85,B 0,C 180,E1 34465.43,E2 34465.43} C_VEL
LIN {X 0,Y 727.916,Z 1196.957,A -85,B 0,C 180,E1 34463.374,E2 34463.374} C_VEL
LIN {X 0,Y 727.936,Z 1191.148,A -85,B 0,C 180,E1 34461.31,E2 34461.31} C_VEL
LIN {X 0,Y 727.945,Z 1183.638,A -85,B 0,C 180,E1 34459.234,E2 34459.234} C_VEL
LIN {X 0,Y 728.028,Z 1173.527,A -85,B 0,C 180,E1 34456.983,E2 34456.983} C_VEL
LIN {X 0,Y 728.084,Z 1164.528,A -85,B 0,C 180,E1 34455.282,E2 34455.282} C_VEL
LIN {X 0,Y 728.169,Z 1154.741,A -85,B 0,C 180,E1 34453.651,E2 34453.651} C_VEL
LIN {X 0,Y 728.298,Z 1144.115,A -85,B 0,C 180,E1 34452.07,E2 34452.07} C_VEL
LIN {X 0,Y 728.489,Z 1130.976,A -85,B 0,C 180,E1 34450.318,E2 34450.318} C_VEL
LIN {X 0,Y 728.74,Z 1113.473,A -85,B 0,C 180,E1 34448.265,E2 34448.265} C_VEL
LIN {X 0,Y 728.955,Z 1098.834,A -85,B 0,C 180,E1 34446.732,E2 34446.732} C_VEL
LIN {X 0,Y 729.277,Z 1082.529,A -85,B 0,C 180,E1 34445.183,E2 34445.183} C_VEL
LIN {X 0,Y 729.687,Z 1061.274,A -85,B 0,C 180,E1 34443.38,E2 34443.38} C_VEL
LIN {X 0,Y 730.038,Z 1043.447,A -85,B 0,C 180,E1 34442.025,E2 34442.025} C_VEL
LIN {X 0,Y 730.495,Z 1023.598,A -85,B 0,C 180,E1 34440.659,E2 34440.659} C_VEL
LIN {X 0,Y 731.013,Z 999.732,A -85,B 0,C 180,E1 34439.204,E2 34439.204} C_VEL
LIN {X 0,Y 731.426,Z 978.537,A -85,B 0,C 180,E1 34438.06,E2 34438.06} C_VEL
LIN {X 0,Y 731.862,Z 957.721,A -85,B 0,C 180,E1 34437.061,E2 34437.061} C_VEL
LIN {X 0,Y 732.438,Z 932.735,A -85,B 0,C 180,E1 34436.013,E2 34436.013} C_VEL
LIN {X 0,Y 732.844,Z 907.028,A -85,B 0,C 180,E1 34435.109,E2 34435.109} C_VEL
LIN {X 0,Y 733.216,Z 883.776,A -85,B 0,C 180,E1 34434.416,E2 34434.416} C_VEL
LIN {X 0,Y 733.575,Z 857.309,A -85,B 0,C 180,E1 34433.785,E2 34433.785} C_VEL
LIN {X 0,Y 733.855,Z 829.91,A -85,B 0,C 180,E1 34433.298,E2 34433.298} C_VEL
LIN {X 0,Y 734.293,Z 733.648,A -85,B 0,C 180,E1 34432.137,E2 34432.137} C_VEL
LIN {X 0,Y 735.2,Z 510.797,A -85,B 0,C 180,E1 34429.44,E2 34429.44} C_VEL
LIN {X 0,Y 735.739,Z 358.813,A -85,B 0,C 180,E1 34427.536,E2 34427.536} C_VEL
LIN {X 0,Y 733.577,Z 350.268,A -85,B 0,C 180,E1 34427.253,E2 34427.253} C_VEL
LIN {X 0,Y 733.823,Z 326.428,A -85,B 0,C 180,E1 34425.655,E2 34425.655} C_VEL
LIN {X 0,Y 729.134,Z 316.486,A -85,B 0,C 180,E1 34424.598,E2 34424.598} C_VEL
LIN {X 0,Y 728.148,Z 313.533,A -85,B 0,C 180,E1 34424.293,E2 34424.293} C_VEL
LIN {X 0,Y 728.124,Z 313.523,A -85,B 0,C 180,E1 34421.43,E2 34421.43} C_VEL
LIN {X 0,Y 728.157,Z 313.524,A -85,B 0,C 180,E1 34418.567,E2 34418.567} C_VEL
LIN {X 0,Y 728.135,Z 313.53,A -85,B 0,C 180,E1 34415.512,E2 34415.512} C_VEL
LIN {X 0,Y 728.133,Z 313.523,A -85,B 0,C 180,E1 34412.662,E2 34412.662} C_VEL
LIN {X 0,Y 728.158,Z 313.524,A -85,B 0,C 180,E1 34409.627,E2 34409.627} C_VEL
LIN {X 0,Y 728.113,Z 313.525,A -85,B 0,C 180,E1 34406.771,E2 34406.771} C_VEL
LIN {X 0,Y 728.154,Z 313.522,A -85,B 0,C 180,E1 34403.897,E2 34403.897} C_VEL
LIN {X 0,Y 728.116,Z 313.523,A -85,B 0,C 180,E1 34401.088,E2 34401.088} C_VEL
LIN {X 0,Y 728.121,Z 313.524,A -85,B 0,C 180,E1 34398.329,E2 34398.329} C_VEL
LIN {X 0,Y 728.146,Z 313.523,A -85,B 0,C 180,E1 34395.287,E2 34395.287} C_VEL
LIN {X 0,Y 728.099,Z 313.528,A -85,B 0,C 180,E1 34392.532,E2 34392.532} C_VEL
LIN {X 0,Y 728.159,Z 313.521,A -85,B 0,C 180,E1 34389.724,E2 34389.724} C_VEL
LIN {X 0,Y 728.106,Z 313.531,A -85,B 0,C 180,E1 34386.783,E2 34386.783} C_VEL
LIN {X 0,Y 728.097,Z 313.524,A -85,B 0,C 180,E1 34384.174,E2 34384.174} C_VEL
LIN {X 0,Y 728.161,Z 313.526,A -85,B 0,C 180,E1 34381.259,E2 34381.259} C_VEL
LIN {X 0,Y 728.092,Z 313.527,A -85,B 0,C 180,E1 34378.505,E2 34378.505} C_VEL
LIN {X 0,Y 728.089,Z 313.524,A -85,B 0,C 180,E1 34375.984,E2 34375.984} C_VEL
LIN {X 0,Y 728.163,Z 313.531,A -85,B 0,C 180,E1 34373.104,E2 34373.104} C_VEL
LIN {X 0,Y 728.082,Z 313.527,A -85,B 0,C 180,E1 34370.275,E2 34370.275} C_VEL
LIN {X 0,Y 728.078,Z 313.53,A -85,B 0,C 180,E1 34367.871,E2 34367.871} C_VEL
LIN {X 0,Y 728.087,Z 313.527,A -85,B 0,C 180,E1 34366.337,E2 34366.337} C_VEL
LIN {X 0,Y 727.057,Z 313.654,A -85,B 0,C 180,E1 34365.731,E2 34365.731} C_VEL
LIN {X 0,Y 720.646,Z 314.454,A -85,B 0,C 180,E1 34364.033,E2 34364.033} C_VEL
LIN {X 0,Y 720.146,Z 314.516,A -85,B 0,C 180,E1 34363.591,E2 34363.591} C_VEL
LIN {X 0,Y 720.195,Z 314.513,A -85,B 0,C 180,E1 34360.621,E2 34360.621} C_VEL
LIN {X 0,Y 720.131,Z 314.521,A -85,B 0,C 180,E1 34357.982,E2 34357.982} C_VEL
LIN {X 0,Y 720.126,Z 314.519,A -85,B 0,C 180,E1 34355.619,E2 34355.619} C_VEL
LIN {X 0,Y 720.176,Z 314.515,A -85,B 0,C 180,E1 34352.999,E2 34352.999} C_VEL
LIN {X 0,Y 720.136,Z 314.513,A -85,B 0,C 180,E1 34350.01,E2 34350.01} C_VEL
LIN {X 0,Y 720.116,Z 314.524,A -85,B 0,C 180,E1 34347.585,E2 34347.585} C_VEL
LIN {X 0,Y 720.123,Z 314.514,A -85,B 0,C 180,E1 34345.203,E2 34345.203} C_VEL
LIN {X 0,Y 720.196,Z 314.514,A -85,B 0,C 180,E1 34342.311,E2 34342.311} C_VEL
LIN {X 0,Y 720.112,Z 314.526,A -85,B 0,C 180,E1 34339.576,E2 34339.576} C_VEL
LIN {X 0,Y 720.108,Z 314.525,A -85,B 0,C 180,E1 34337.265,E2 34337.265} C_VEL
LIN {X 0,Y 720.133,Z 314.529,A -85,B 0,C 180,E1 34334.856,E2 34334.856} C_VEL
LIN {X 0,Y 720.224,Z 314.697,A -85,B 0,C 180,E1 34334.13,E2 34334.13} C_VEL
LIN {X 0,Y 721.514,Z 318.104,A -85,B 0,C 180,E1 34333.779,E2 34333.779} C_VEL
LIN {X 0,Y 723.027,Z 321.575,A -85,B 0,C 180,E1 34333.445,E2 34333.445} C_VEL
LIN {X 0,Y 729.776,Z 331.97,A -85,B 0,C 180,E1 34332.807,E2 34332.807} C_VEL
LIN {X 0,Y 729.13,Z 474.606,A -85,B 0,C 180,E1 34331.003,E2 34331.003} C_VEL
LIN {X 0,Y 728.025,Z 691.305,A -85,B 0,C 180,E1 34328.355,E2 34328.355} C_VEL
LIN {X 0,Y 727.422,Z 799.793,A -85,B 0,C 180,E1 34327.038,E2 34327.038} C_VEL
LIN {X 0,Y 727.08,Z 827.04,A -85,B 0,C 180,E1 34326.552,E2 34326.552} C_VEL
LIN {X 0,Y 726.622,Z 853.457,A -85,B 0,C 180,E1 34325.921,E2 34325.921} C_VEL
LIN {X 0,Y 726.155,Z 876.429,A -85,B 0,C 180,E1 34325.235,E2 34325.235} C_VEL
LIN {X 0,Y 725.657,Z 901.575,A -85,B 0,C 180,E1 34324.349,E2 34324.349} C_VEL
LIN {X 0,Y 724.981,Z 926.779,A -85,B 0,C 180,E1 34323.292,E2 34323.292} C_VEL
LIN {X 0,Y 724.407,Z 947.684,A -85,B 0,C 180,E1 34322.286,E2 34322.286} C_VEL
LIN {X 0,Y 723.861,Z 967.868,A -85,B 0,C 180,E1 34321.197,E2 34321.197} C_VEL
LIN {X 0,Y 723.287,Z 991.604,A -85,B 0,C 180,E1 34319.754,E2 34319.754} C_VEL
LIN {X 0,Y 722.688,Z 1012.24,A -85,B 0,C 180,E1 34318.33,E2 34318.33} C_VEL
LIN {X 0,Y 722.192,Z 1030.092,A -85,B 0,C 180,E1 34316.969,E2 34316.969} C_VEL
LIN {X 0,Y 721.754,Z 1050.317,A -85,B 0,C 180,E1 34315.257,E2 34315.257} C_VEL
LIN {X 0,Y 721.296,Z 1067.625,A -85,B 0,C 180,E1 34313.608,E2 34313.608} C_VEL
LIN {X 0,Y 720.987,Z 1082.214,A -85,B 0,C 180,E1 34312.075,E2 34312.075} C_VEL
LIN {X 0,Y 720.692,Z 1098.252,A -85,B 0,C 180,E1 34310.209,E2 34310.209} C_VEL
LIN {X 0,Y 720.444,Z 1112.781,A -85,B 0,C 180,E1 34308.279,E2 34308.279} C_VEL
LIN {X 0,Y 720.269,Z 1123.938,A -85,B 0,C 180,E1 34306.616,E2 34306.616} C_VEL
LIN {X 0,Y 720.132,Z 1133.81,A -85,B 0,C 180,E1 34304.966,E2 34304.966} C_VEL
LIN {X 0,Y 720.059,Z 1142.481,A -85,B 0,C 180,E1 34303.327,E2 34303.327} C_VEL
LIN {X 0,Y 719.996,Z 1150.736,A -85,B 0,C 180,E1 34301.535,E2 34301.535} C_VEL
LIN {X 0,Y 719.951,Z 1158.601,A -85,B 0,C 180,E1 34299.513,E2 34299.513} C_VEL
LIN {X 0,Y 719.925,Z 1165.229,A -85,B 0,C 180,E1 34297.341,E2 34297.341} C_VEL
LIN {X 0,Y 719.912,Z 1169.958,A -85,B 0,C 180,E1 34295.259,E2 34295.259} C_VEL
LIN {X 0,Y 719.912,Z 1173.231,A -85,B 0,C 180,E1 34293.105,E2 34293.105} C_VEL
LIN {X 0,Y 719.912,Z 1174.702,A -85,B 0,C 180,E1 34291.035,E2 34291.035} C_VEL
LIN {X 0,Y 719.895,Z 1174.817,A -85,B 0,C 180,E1 34289.284,E2 34289.284} C_VEL
LIN {X 0,Y 719.906,Z 1173.793,A -85,B 0,C 180,E1 34287.373,E2 34287.373} C_VEL
LIN {X 0,Y 719.909,Z 1170.999,A -85,B 0,C 180,E1 34285.22,E2 34285.22} C_VEL
LIN {X 0,Y 719.917,Z 1166.48,A -85,B 0,C 180,E1 34283.06,E2 34283.06} C_VEL
LIN {X 0,Y 719.939,Z 1160.779,A -85,B 0,C 180,E1 34281.052,E2 34281.052} C_VEL
LIN {X 0,Y 719.978,Z 1152.859,A -85,B 0,C 180,E1 34278.87,E2 34278.87} C_VEL
LIN {X 0,Y 720.052,Z 1143.343,A -85,B 0,C 180,E1 34276.755,E2 34276.755} C_VEL
LIN {X 0,Y 720.126,Z 1134.318,A -85,B 0,C 180,E1 34275.034,E2 34275.034} C_VEL
LIN {X 0,Y 720.261,Z 1124.503,A -85,B 0,C 180,E1 34273.383,E2 34273.383} C_VEL
LIN {X 0,Y 720.434,Z 1113.14,A -85,B 0,C 180,E1 34271.682,E2 34271.682} C_VEL
LIN {X 0,Y 720.688,Z 1098.256,A -85,B 0,C 180,E1 34269.701,E2 34269.701} C_VEL
LIN {X 0,Y 720.98,Z 1082.253,A -85,B 0,C 180,E1 34267.839,E2 34267.839} C_VEL
LIN {X 0,Y 721.293,Z 1067.571,A -85,B 0,C 180,E1 34266.297,E2 34266.297} C_VEL
LIN {X 0,Y 721.776,Z 1048.956,A -85,B 0,C 180,E1 34264.529,E2 34264.529} C_VEL
LIN {X 0,Y 722.209,Z 1029.597,A -85,B 0,C 180,E1 34262.902,E2 34262.902} C_VEL
LIN {X 0,Y 722.706,Z 1011.634,A -85,B 0,C 180,E1 34261.536,E2 34261.536} C_VEL
LIN {X 0,Y 723.349,Z 989.529,A -85,B 0,C 180,E1 34260.021,E2 34260.021} C_VEL
LIN {X 0,Y 723.879,Z 967.024,A -85,B 0,C 180,E1 34258.665,E2 34258.665} C_VEL
LIN {X 0,Y 724.442,Z 946.726,A -85,B 0,C 180,E1 34257.575,E2 34257.575} C_VEL
LIN {X 0,Y 725.094,Z 923.671,A -85,B 0,C 180,E1 34256.478,E2 34256.478} C_VEL
LIN {X 0,Y 725.703,Z 897.608,A -85,B 0,C 180,E1 34255.414,E2 34255.414} C_VEL
LIN {X 0,Y 726.165,Z 875.494,A -85,B 0,C 180,E1 34254.645,E2 34254.645} C_VEL
LIN {X 0,Y 726.632,Z 852.584,A -85,B 0,C 180,E1 34253.966,E2 34253.966} C_VEL
LIN {X 0,Y 727.114,Z 825.634,A -85,B 0,C 180,E1 34253.329,E2 34253.329} C_VEL
LIN {X 0,Y 727.441,Z 798.301,A -85,B 0,C 180,E1 34252.85,E2 34252.85} C_VEL
LIN {X 0,Y 728.673,Z 564.02,A -85,B 0,C 180,E1 34250.011,E2 34250.011} C_VEL
LIN {X 0,Y 729.738,Z 358.517,A -85,B 0,C 180,E1 34247.448,E2 34247.448} C_VEL
LIN {X 0,Y 729.684,Z 331.572,A -85,B 0,C 180,E1 34247.091,E2 34247.091} C_VEL
LIN {X 0,Y 722.598,Z 320.887,A -85,B 0,C 180,E1 34246.418,E2 34246.418} C_VEL
LIN {X 0,Y 720.219,Z 314.529,A -85,B 0,C 180,E1 34245.767,E2 34245.767} C_VEL
LIN {X 0,Y 720.13,Z 314.524,A -85,B 0,C 180,E1 34242.97,E2 34242.97} C_VEL
LIN {X 0,Y 720.116,Z 314.525,A -85,B 0,C 180,E1 34240.581,E2 34240.581} C_VEL
LIN {X 0,Y 720.125,Z 314.525,A -85,B 0,C 180,E1 34238.2,E2 34238.2} C_VEL
LIN {X 0,Y 720.183,Z 314.514,A -85,B 0,C 180,E1 34235.28,E2 34235.28} C_VEL
LIN {X 0,Y 720.11,Z 314.525,A -85,B 0,C 180,E1 34232.563,E2 34232.563} C_VEL
LIN {X 0,Y 720.11,Z 314.514,A -85,B 0,C 180,E1 34230.267,E2 34230.267} C_VEL
LIN {X 0,Y 720.131,Z 314.524,A -85,B 0,C 180,E1 34227.899,E2 34227.899} C_VEL
LIN {X 0,Y 720.164,Z 314.519,A -85,B 0,C 180,E1 34224.878,E2 34224.878} C_VEL
LIN {X 0,Y 720.123,Z 314.521,A -85,B 0,C 180,E1 34222.362,E2 34222.362} C_VEL
LIN {X 0,Y 720.122,Z 314.511,A -85,B 0,C 180,E1 34220.057,E2 34220.057} C_VEL
LIN {X 0,Y 720.166,Z 314.522,A -85,B 0,C 180,E1 34217.483,E2 34217.483} C_VEL
LIN {X 0,Y 720.154,Z 314.512,A -85,B 0,C 180,E1 34214.473,E2 34214.473} C_VEL
LIN {X 0,Y 720.132,Z 314.521,A -85,B 0,C 180,E1 34212.021,E2 34212.021} C_VEL
LIN {X 0,Y 720.144,Z 314.517,A -85,B 0,C 180,E1 34209.591,E2 34209.591} C_VEL
LIN {X 0,Y 720.218,Z 314.517,A -85,B 0,C 180,E1 34206.697,E2 34206.697} C_VEL
LIN {X 0,Y 720.142,Z 314.514,A -85,B 0,C 180,E1 34203.901,E2 34203.901} C_VEL
LIN {X 0,Y 720.151,Z 314.514,A -85,B 0,C 180,E1 34201.432,E2 34201.432} C_VEL
LIN {X 0,Y 720.222,Z 314.512,A -85,B 0,C 180,E1 34198.568,E2 34198.568} C_VEL
LIN {X 0,Y 720.15,Z 314.511,A -85,B 0,C 180,E1 34195.7,E2 34195.7} C_VEL
LIN {X 0,Y 720.168,Z 314.521,A -85,B 0,C 180,E1 34193.142,E2 34193.142} C_VEL
LIN {X 0,Y 720.201,Z 314.509,A -85,B 0,C 180,E1 34190.087,E2 34190.087} C_VEL
LIN {X 0,Y 720.158,Z 314.518,A -85,B 0,C 180,E1 34187.328,E2 34187.328} C_VEL
LIN {X 0,Y 720.221,Z 314.51,A -85,B 0,C 180,E1 34184.541,E2 34184.541} C_VEL
LIN {X 0,Y 720.172,Z 314.515,A -85,B 0,C 180,E1 34181.545,E2 34181.545} C_VEL
LIN {X 0,Y 720.179,Z 314.511,A -85,B 0,C 180,E1 34178.839,E2 34178.839} C_VEL
LIN {X 0,Y 720.218,Z 314.506,A -85,B 0,C 180,E1 34175.823,E2 34175.823} C_VEL
LIN {X 0,Y 720.17,Z 314.517,A -85,B 0,C 180,E1 34172.999,E2 34172.999} C_VEL
LIN {X 0,Y 720.217,Z 314.511,A -85,B 0,C 180,E1 34170.189,E2 34170.189} C_VEL
LIN {X 0,Y 720.184,Z 314.513,A -85,B 0,C 180,E1 34167.216,E2 34167.216} C_VEL
LIN {X 0,Y 720.214,Z 314.521,A -85,B 0,C 180,E1 34164.306,E2 34164.306} C_VEL
LIN {X 0,Y 720.203,Z 314.514,A -85,B 0,C 180,E1 34161.234,E2 34161.234} C_VEL
LIN {X 0,Y 720.201,Z 314.524,A -85,B 0,C 180,E1 34158.316,E2 34158.316} C_VEL
LIN {X 0,Y 720.219,Z 314.627,A -85,B 0,C 180,E1 34156.26,E2 34156.26} C_VEL
LIN {X 0,Y 721.485,Z 317.954,A -85,B 0,C 180,E1 34155.916,E2 34155.916} C_VEL
LIN {X 0,Y 727.499,Z 330.947,A -85,B 0,C 180,E1 34154.519,E2 34154.519} C_VEL
LIN {X 0,Y 727.216,Z 351.094,A -85,B 0,C 180,E1 34153.184,E2 34153.184} C_VEL
LIN {X 0,Y 729.917,Z 362.046,A -85,B 0,C 180,E1 34152.841,E2 34152.841} C_VEL
LIN {X 0,Y 728.768,Z 574.71,A -85,B 0,C 180,E1 34150.181,E2 34150.181} C_VEL
LIN {X 0,Y 727.655,Z 798.989,A -85,B 0,C 180,E1 34147.47,E2 34147.47} C_VEL
LIN {X 0,Y 727.387,Z 835.164,A -85,B 0,C 180,E1 34147.001,E2 34147.001} C_VEL
LIN {X 0,Y 726.978,Z 862.471,A -85,B 0,C 180,E1 34146.48,E2 34146.48} C_VEL
LIN {X 0,Y 726.542,Z 888.181,A -85,B 0,C 180,E1 34145.837,E2 34145.837} C_VEL
LIN {X 0,Y 725.973,Z 916.212,A -85,B 0,C 180,E1 34144.956,E2 34144.956} C_VEL
LIN {X 0,Y 725.376,Z 939.909,A -85,B 0,C 180,E1 34144.06,E2 34144.06} C_VEL
LIN {X 0,Y 724.836,Z 961.083,A -85,B 0,C 180,E1 34143.139,E2 34143.139} C_VEL
LIN {X 0,Y 724.298,Z 983.24,A -85,B 0,C 180,E1 34142.045,E2 34142.045} C_VEL
LIN {X 0,Y 723.606,Z 1008.626,A -85,B 0,C 180,E1 34140.609,E2 34140.609} C_VEL
LIN {X 0,Y 723.047,Z 1028.239,A -85,B 0,C 180,E1 34139.355,E2 34139.355} C_VEL
LIN {X 0,Y 722.54,Z 1047.296,A -85,B 0,C 180,E1 34138.005,E2 34138.005} C_VEL
LIN {X 0,Y 721.988,Z 1069.76,A -85,B 0,C 180,E1 34136.217,E2 34136.217} C_VEL
LIN {X 0,Y 721.543,Z 1086.385,A -85,B 0,C 180,E1 34134.739,E2 34134.739} C_VEL
LIN {X 0,Y 721.208,Z 1103.097,A -85,B 0,C 180,E1 34133.1,E2 34133.1} C_VEL
LIN {X 0,Y 720.819,Z 1120.837,A -85,B 0,C 180,E1 34131.14,E2 34131.14} C_VEL
LIN {X 0,Y 720.582,Z 1133.807,A -85,B 0,C 180,E1 34129.536,E2 34129.536} C_VEL
LIN {X 0,Y 720.389,Z 1146.004,A -85,B 0,C 180,E1 34127.863,E2 34127.863} C_VEL
LIN {X 0,Y 720.214,Z 1158.903,A -85,B 0,C 180,E1 34125.872,E2 34125.872} C_VEL
LIN {X 0,Y 720.078,Z 1170.244,A -85,B 0,C 180,E1 34123.817,E2 34123.817} C_VEL
LIN {X 0,Y 719.995,Z 1178.432,A -85,B 0,C 180,E1 34122.104,E2 34122.104} C_VEL
LIN {X 0,Y 719.965,Z 1186.135,A -85,B 0,C 180,E1 34120.239,E2 34120.239} C_VEL
LIN {X 0,Y 719.933,Z 1193.544,A -85,B 0,C 180,E1 34118.001,E2 34118.001} C_VEL
LIN {X 0,Y 719.918,Z 1198.937,A -85,B 0,C 180,E1 34115.819,E2 34115.819} C_VEL
LIN {X 0,Y 719.909,Z 1202.484,A -85,B 0,C 180,E1 34113.743,E2 34113.743} C_VEL
LIN {X 0,Y 719.909,Z 1204.549,A -85,B 0,C 180,E1 34111.592,E2 34111.592} C_VEL
LIN {X 0,Y 719.89,Z 1204.872,A -85,B 0,C 180,E1 34109.523,E2 34109.523} C_VEL
LIN {X 0,Y 719.906,Z 1203.902,A -85,B 0,C 180,E1 34107.532,E2 34107.532} C_VEL
LIN {X 0,Y 719.908,Z 1201.178,A -85,B 0,C 180,E1 34105.38,E2 34105.38} C_VEL
LIN {X 0,Y 719.917,Z 1196.832,A -85,B 0,C 180,E1 34103.249,E2 34103.249} C_VEL
LIN {X 0,Y 719.937,Z 1190.891,A -85,B 0,C 180,E1 34101.132,E2 34101.132} C_VEL
LIN {X 0,Y 719.972,Z 1183.001,A -85,B 0,C 180,E1 34098.951,E2 34098.951} C_VEL
LIN {X 0,Y 720.061,Z 1173.152,A -85,B 0,C 180,E1 34096.762,E2 34096.762} C_VEL
LIN {X 0,Y 720.128,Z 1164.064,A -85,B 0,C 180,E1 34095.034,E2 34095.034} C_VEL
LIN {X 0,Y 720.263,Z 1154.221,A -85,B 0,C 180,E1 34093.383,E2 34093.383} C_VEL
LIN {X 0,Y 720.441,Z 1142.511,A -85,B 0,C 180,E1 34091.637,E2 34091.637} C_VEL
LIN {X 0,Y 720.722,Z 1126.521,A -85,B 0,C 180,E1 34089.537,E2 34089.537} C_VEL
LIN {X 0,Y 720.991,Z 1111.843,A -85,B 0,C 180,E1 34087.839,E2 34087.839} C_VEL
LIN {X 0,Y 721.307,Z 1097.128,A -85,B 0,C 180,E1 34086.297,E2 34086.297} C_VEL
LIN {X 0,Y 721.785,Z 1077.881,A -85,B 0,C 180,E1 34084.481,E2 34084.481} C_VEL
LIN {X 0,Y 722.23,Z 1059.06,A -85,B 0,C 180,E1 34082.905,E2 34082.905} C_VEL
LIN {X 0,Y 722.736,Z 1041.03,A -85,B 0,C 180,E1 34081.537,E2 34081.537} C_VEL
LIN {X 0,Y 723.365,Z 1018.082,A -85,B 0,C 180,E1 34079.976,E2 34079.976} C_VEL
LIN {X 0,Y 723.901,Z 996.241,A -85,B 0,C 180,E1 34078.666,E2 34078.666} C_VEL
LIN {X 0,Y 724.472,Z 975.869,A -85,B 0,C 180,E1 34077.576,E2 34077.576} C_VEL
LIN {X 0,Y 725.163,Z 951.713,A -85,B 0,C 180,E1 34076.434,E2 34076.434} C_VEL
LIN {X 0,Y 725.714,Z 926.414,A -85,B 0,C 180,E1 34075.415,E2 34075.415} C_VEL
LIN {X 0,Y 726.174,Z 904.863,A -85,B 0,C 180,E1 34074.67,E2 34074.67} C_VEL
LIN {X 0,Y 726.646,Z 881.764,A -85,B 0,C 180,E1 34073.988,E2 34073.988} C_VEL
LIN {X 0,Y 727.127,Z 854.692,A -85,B 0,C 180,E1 34073.354,E2 34073.354} C_VEL
LIN {X 0,Y 727.448,Z 827.377,A -85,B 0,C 180,E1 34072.882,E2 34072.882} C_VEL
LIN {X 0,Y 728.656,Z 595.56,A -85,B 0,C 180,E1 34070.074,E2 34070.074} C_VEL
LIN {X 0,Y 729.77,Z 388.001,A -85,B 0,C 180,E1 34067.489,E2 34067.489} C_VEL
LIN {X 0,Y 729.748,Z 360.674,A -85,B 0,C 180,E1 34067.129,E2 34067.129} C_VEL
LIN {X 0,Y 727.105,Z 350.268,A -85,B 0,C 180,E1 34066.779,E2 34066.779} C_VEL
LIN {X 0,Y 727.452,Z 330.61,A -85,B 0,C 180,E1 34065.454,E2 34065.454} C_VEL
LIN {X 0,Y 721.485,Z 317.954,A -85,B 0,C 180,E1 34064.084,E2 34064.084} C_VEL
LIN {X 0,Y 720.202,Z 314.524,A -85,B 0,C 180,E1 34063.706,E2 34063.706} C_VEL
LIN {X 0,Y 720.209,Z 314.503,A -85,B 0,C 180,E1 34060.732,E2 34060.732} C_VEL
LIN {X 0,Y 720.204,Z 314.512,A -85,B 0,C 180,E1 34057.653,E2 34057.653} C_VEL
LIN {X 0,Y 720.194,Z 314.512,A -85,B 0,C 180,E1 34054.726,E2 34054.726} C_VEL
LIN {X 0,Y 720.214,Z 314.521,A -85,B 0,C 180,E1 34051.654,E2 34051.654} C_VEL
LIN {X 0,Y 720.175,Z 314.513,A -85,B 0,C 180,E1 34048.802,E2 34048.802} C_VEL
LIN {X 0,Y 720.215,Z 314.515,A -85,B 0,C 180,E1 34045.933,E2 34045.933} C_VEL
LIN {X 0,Y 720.174,Z 314.519,A -85,B 0,C 180,E1 34043.05,E2 34043.05} C_VEL
LIN {X 0,Y 720.19,Z 314.505,A -85,B 0,C 180,E1 34040.31,E2 34040.31} C_VEL
LIN {X 0,Y 720.193,Z 314.52,A -85,B 0,C 180,E1 34037.201,E2 34037.201} C_VEL
LIN {X 0,Y 720.164,Z 314.508,A -85,B 0,C 180,E1 34034.473,E2 34034.473} C_VEL
LIN {X 0,Y 720.22,Z 314.516,A -85,B 0,C 180,E1 34031.613,E2 34031.613} C_VEL
LIN {X 0,Y 720.164,Z 314.513,A -85,B 0,C 180,E1 34028.785,E2 34028.785} C_VEL
LIN {X 0,Y 720.166,Z 314.516,A -85,B 0,C 180,E1 34026.137,E2 34026.137} C_VEL
LIN {X 0,Y 720.216,Z 314.509,A -85,B 0,C 180,E1 34023.183,E2 34023.183} C_VEL
LIN {X 0,Y 720.15,Z 314.519,A -85,B 0,C 180,E1 34020.398,E2 34020.398} C_VEL
LIN {X 0,Y 720.173,Z 314.511,A -85,B 0,C 180,E1 34017.772,E2 34017.772} C_VEL
LIN {X 0,Y 720.17,Z 314.522,A -85,B 0,C 180,E1 34014.662,E2 34014.662} C_VEL
LIN {X 0,Y 720.141,Z 314.514,A -85,B 0,C 180,E1 34012.099,E2 34012.099} C_VEL
LIN {X 0,Y 720.182,Z 314.512,A -85,B 0,C 180,E1 34009.44,E2 34009.44} C_VEL
LIN {X 0,Y 720.157,Z 314.515,A -85,B 0,C 180,E1 34006.429,E2 34006.429} C_VEL
LIN {X 0,Y 720.134,Z 314.517,A -85,B 0,C 180,E1 34003.903,E2 34003.903} C_VEL
LIN {X 0,Y 720.146,Z 314.516,A -85,B 0,C 180,E1 34003.591,E2 34003.591} C_VEL
LIN {X 0,Y 719.208,Z 314.642,A -85,B 0,C 180,E1 34002.979,E2 34002.979} C_VEL
LIN {X 0,Y 712.835,Z 315.443,A -85,B 0,C 180,E1 34001.262,E2 34001.262} C_VEL
LIN {X 0,Y 712.28,Z 315.503,A -85,B 0,C 180,E1 34000.816,E2 34000.816} C_VEL
LIN {X 0,Y 712.197,Z 315.51,A -85,B 0,C 180,E1 33998.071,E2 33998.071} C_VEL
LIN {X 0,Y 712.186,Z 315.508,A -85,B 0,C 180,E1 33995.664,E2 33995.664} C_VEL
LIN {X 0,Y 712.219,Z 315.504,A -85,B 0,C 180,E1 33993.124,E2 33993.124} C_VEL
LIN {X 0,Y 712.207,Z 315.5,A -85,B 0,C 180,E1 33990.106,E2 33990.106} C_VEL
LIN {X 0,Y 712.178,Z 315.513,A -85,B 0,C 180,E1 33987.661,E2 33987.661} C_VEL
LIN {X 0,Y 712.177,Z 315.502,A -85,B 0,C 180,E1 33985.346,E2 33985.346} C_VEL
LIN {X 0,Y 712.249,Z 315.51,A -85,B 0,C 180,E1 33982.613,E2 33982.613} C_VEL
LIN {X 0,Y 712.187,Z 315.515,A -85,B 0,C 180,E1 33979.772,E2 33979.772} C_VEL
LIN {X 0,Y 712.169,Z 315.515,A -85,B 0,C 180,E1 33977.364,E2 33977.364} C_VEL
LIN {X 0,Y 712.18,Z 315.519,A -85,B 0,C 180,E1 33975.039,E2 33975.039} C_VEL
LIN {X 0,Y 712.213,Z 315.545,A -85,B 0,C 180,E1 33974.695,E2 33974.695} C_VEL
LIN {X 0,Y 713.356,Z 318.666,A -85,B 0,C 180,E1 33974.369,E2 33974.369} C_VEL
LIN {X 0,Y 714.644,Z 321.523,A -85,B 0,C 180,E1 33974.087,E2 33974.087} C_VEL
LIN {X 0,Y 723.946,Z 335.615,A -85,B 0,C 180,E1 33973.188,E2 33973.188} C_VEL
LIN {X 0,Y 722.746,Z 529.54,A -85,B 0,C 180,E1 33970.735,E2 33970.735} C_VEL
LIN {X 0,Y 721.371,Z 757.055,A -85,B 0,C 180,E1 33967.957,E2 33967.957} C_VEL
LIN {X 0,Y 720.994,Z 802.607,A -85,B 0,C 180,E1 33967.38,E2 33967.38} C_VEL
LIN {X 0,Y 720.541,Z 829.98,A -85,B 0,C 180,E1 33966.872,E2 33966.872} C_VEL
LIN {X 0,Y 720.021,Z 855.319,A -85,B 0,C 180,E1 33966.249,E2 33966.249} C_VEL
LIN {X 0,Y 719.438,Z 880.123,A -85,B 0,C 180,E1 33965.491,E2 33965.491} C_VEL
LIN {X 0,Y 718.729,Z 906.201,A -85,B 0,C 180,E1 33964.534,E2 33964.534} C_VEL
LIN {X 0,Y 718.016,Z 928.781,A -85,B 0,C 180,E1 33963.562,E2 33963.562} C_VEL
LIN {X 0,Y 717.344,Z 949.478,A -85,B 0,C 180,E1 33962.549,E2 33962.549} C_VEL
LIN {X 0,Y 716.641,Z 972.696,A -85,B 0,C 180,E1 33961.266,E2 33961.266} C_VEL
LIN {X 0,Y 715.871,Z 995.605,A -85,B 0,C 180,E1 33959.817,E2 33959.817} C_VEL
LIN {X 0,Y 715.251,Z 1014.062,A -85,B 0,C 180,E1 33958.515,E2 33958.515} C_VEL
LIN {X 0,Y 714.638,Z 1032.936,A -85,B 0,C 180,E1 33957.046,E2 33957.046} C_VEL
LIN {X 0,Y 714.041,Z 1053.687,A -85,B 0,C 180,E1 33955.229,E2 33955.229} C_VEL
LIN {X 0,Y 713.573,Z 1069.252,A -85,B 0,C 180,E1 33953.712,E2 33953.712} C_VEL
LIN {X 0,Y 713.183,Z 1085.33,A -85,B 0,C 180,E1 33951.983,E2 33951.983} C_VEL
LIN {X 0,Y 712.787,Z 1102.181,A -85,B 0,C 180,E1 33949.93,E2 33949.93} C_VEL
LIN {X 0,Y 712.528,Z 1114.533,A -85,B 0,C 180,E1 33948.236,E2 33948.236} C_VEL
LIN {X 0,Y 712.32,Z 1125.753,A -85,B 0,C 180,E1 33946.516,E2 33946.516} C_VEL
LIN {X 0,Y 712.181,Z 1137.517,A -85,B 0,C 180,E1 33944.472,E2 33944.472} C_VEL
LIN {X 0,Y 712.04,Z 1147.88,A -85,B 0,C 180,E1 33942.324,E2 33942.324} C_VEL
LIN {X 0,Y 711.983,Z 1155.968,A -85,B 0,C 180,E1 33940.355,E2 33940.355} C_VEL
LIN {X 0,Y 711.943,Z 1163.22,A -85,B 0,C 180,E1 33938.155,E2 33938.155} C_VEL
LIN {X 0,Y 711.922,Z 1168.67,A -85,B 0,C 180,E1 33935.965,E2 33935.965} C_VEL
LIN {X 0,Y 711.912,Z 1172.322,A -85,B 0,C 180,E1 33933.865,E2 33933.865} C_VEL
LIN {X 0,Y 711.907,Z 1174.518,A -85,B 0,C 180,E1 33931.61,E2 33931.61} C_VEL
LIN {X 0,Y 711.89,Z 1174.884,A -85,B 0,C 180,E1 33929.517,E2 33929.517} C_VEL
LIN {X 0,Y 711.905,Z 1173.937,A -85,B 0,C 180,E1 33927.505,E2 33927.505} C_VEL
LIN {X 0,Y 711.908,Z 1171.248,A -85,B 0,C 180,E1 33925.328,E2 33925.328} C_VEL
LIN {X 0,Y 711.917,Z 1167.034,A -85,B 0,C 180,E1 33923.212,E2 33923.212} C_VEL
LIN {X 0,Y 711.944,Z 1161.283,A -85,B 0,C 180,E1 33921.113,E2 33921.113} C_VEL
LIN {X 0,Y 711.979,Z 1153.814,A -85,B 0,C 180,E1 33918.989,E2 33918.989} C_VEL
LIN {X 0,Y 712.087,Z 1143.714,A -85,B 0,C 180,E1 33916.679,E2 33916.679} C_VEL
LIN {X 0,Y 712.175,Z 1134.782,A -85,B 0,C 180,E1 33914.946,E2 33914.946} C_VEL
LIN {X 0,Y 712.352,Z 1124.501,A -85,B 0,C 180,E1 33913.193,E2 33913.193} C_VEL
LIN {X 0,Y 712.555,Z 1113.404,A -85,B 0,C 180,E1 33911.511,E2 33911.511} C_VEL
LIN {X 0,Y 712.867,Z 1098.289,A -85,B 0,C 180,E1 33909.473,E2 33909.473} C_VEL
LIN {X 0,Y 713.23,Z 1082.249,A -85,B 0,C 180,E1 33907.585,E2 33907.585} C_VEL
LIN {X 0,Y 713.636,Z 1067.293,A -85,B 0,C 180,E1 33905.999,E2 33905.999} C_VEL
LIN {X 0,Y 714.188,Z 1048.378,A -85,B 0,C 180,E1 33904.188,E2 33904.188} C_VEL
LIN {X 0,Y 714.754,Z 1029.612,A -85,B 0,C 180,E1 33902.598,E2 33902.598} C_VEL
LIN {X 0,Y 715.321,Z 1012.232,A -85,B 0,C 180,E1 33901.26,E2 33901.26} C_VEL
LIN {X 0,Y 716.08,Z 990.234,A -85,B 0,C 180,E1 33899.731,E2 33899.731} C_VEL
LIN {X 0,Y 716.777,Z 966.938,A -85,B 0,C 180,E1 33898.314,E2 33898.314} C_VEL
LIN {X 0,Y 717.454,Z 946.716,A -85,B 0,C 180,E1 33897.22,E2 33897.22} C_VEL
LIN {X 0,Y 718.181,Z 924.66,A -85,B 0,C 180,E1 33896.16,E2 33896.16} C_VEL
LIN {X 0,Y 718.925,Z 898.867,A -85,B 0,C 180,E1 33895.089,E2 33895.089} C_VEL
LIN {X 0,Y 719.494,Z 876.213,A -85,B 0,C 180,E1 33894.292,E2 33894.292} C_VEL
LIN {X 0,Y 720.057,Z 853.152,A -85,B 0,C 180,E1 33893.601,E2 33893.601} C_VEL
LIN {X 0,Y 720.628,Z 826.497,A -85,B 0,C 180,E1 33892.964,E2 33892.964} C_VEL
LIN {X 0,Y 721.029,Z 799.347,A -85,B 0,C 180,E1 33892.48,E2 33892.48} C_VEL
LIN {X 0,Y 722.498,Z 569.545,A -85,B 0,C 180,E1 33889.67,E2 33889.67} C_VEL
LIN {X 0,Y 723.813,Z 361.521,A -85,B 0,C 180,E1 33887.057,E2 33887.057} C_VEL
LIN {X 0,Y 723.799,Z 335.318,A -85,B 0,C 180,E1 33886.707,E2 33886.707} C_VEL
LIN {X 0,Y 714.319,Z 320.859,A -85,B 0,C 180,E1 33885.782,E2 33885.782} C_VEL
LIN {X 0,Y 712.211,Z 315.518,A -85,B 0,C 180,E1 33885.191,E2 33885.191} C_VEL
LIN {X 0,Y 712.18,Z 315.513,A -85,B 0,C 180,E1 33882.698,E2 33882.698} C_VEL
LIN {X 0,Y 712.184,Z 315.515,A -85,B 0,C 180,E1 33880.334,E2 33880.334} C_VEL
LIN {X 0,Y 712.269,Z 315.509,A -85,B 0,C 180,E1 33877.522,E2 33877.522} C_VEL
LIN {X 0,Y 712.178,Z 315.502,A -85,B 0,C 180,E1 33874.752,E2 33874.752} C_VEL
LIN {X 0,Y 712.169,Z 315.514,A -85,B 0,C 180,E1 33872.309,E2 33872.309} C_VEL
LIN {X 0,Y 712.204,Z 315.501,A -85,B 0,C 180,E1 33869.802,E2 33869.802} C_VEL
LIN {X 0,Y 712.202,Z 315.506,A -85,B 0,C 180,E1 33866.763,E2 33866.763} C_VEL
LIN {X 0,Y 712.179,Z 315.508,A -85,B 0,C 180,E1 33864.291,E2 33864.291} C_VEL
LIN {X 0,Y 712.192,Z 315.511,A -85,B 0,C 180,E1 33861.877,E2 33861.877} C_VEL
LIN {X 0,Y 712.272,Z 315.506,A -85,B 0,C 180,E1 33859.007,E2 33859.007} C_VEL
LIN {X 0,Y 712.191,Z 315.506,A -85,B 0,C 180,E1 33856.203,E2 33856.203} C_VEL
LIN {X 0,Y 712.193,Z 315.502,A -85,B 0,C 180,E1 33853.808,E2 33853.808} C_VEL
LIN {X 0,Y 712.28,Z 315.506,A -85,B 0,C 180,E1 33851.006,E2 33851.006} C_VEL
LIN {X 0,Y 712.206,Z 315.5,A -85,B 0,C 180,E1 33848.152,E2 33848.152} C_VEL
LIN {X 0,Y 712.2,Z 315.51,A -85,B 0,C 180,E1 33845.721,E2 33845.721} C_VEL
LIN {X 0,Y 712.265,Z 315.498,A -85,B 0,C 180,E1 33842.977,E2 33842.977} C_VEL
LIN {X 0,Y 712.219,Z 315.507,A -85,B 0,C 180,E1 33840,E2 33840} C_VEL
LIN {X 0,Y 712.212,Z 315.503,A -85,B 0,C 180,E1 33837.425,E2 33837.425} C_VEL
LIN {X 0,Y 712.284,Z 315.506,A -85,B 0,C 180,E1 33834.522,E2 33834.522} C_VEL
LIN {X 0,Y 712.218,Z 315.5,A -85,B 0,C 180,E1 33831.686,E2 33831.686} C_VEL
LIN {X 0,Y 712.23,Z 315.504,A -85,B 0,C 180,E1 33829.075,E2 33829.075} C_VEL
LIN {X 0,Y 712.27,Z 315.493,A -85,B 0,C 180,E1 33826.027,E2 33826.027} C_VEL
LIN {X 0,Y 712.222,Z 315.505,A -85,B 0,C 180,E1 33823.274,E2 33823.274} C_VEL
LIN {X 0,Y 712.279,Z 315.498,A -85,B 0,C 180,E1 33820.482,E2 33820.482} C_VEL
LIN {X 0,Y 712.238,Z 315.505,A -85,B 0,C 180,E1 33817.464,E2 33817.464} C_VEL
LIN {X 0,Y 712.252,Z 315.5,A -85,B 0,C 180,E1 33814.648,E2 33814.648} C_VEL
LIN {X 0,Y 712.257,Z 315.5,A -85,B 0,C 180,E1 33811.49,E2 33811.49} C_VEL
LIN {X 0,Y 712.251,Z 315.507,A -85,B 0,C 180,E1 33808.595,E2 33808.595} C_VEL
LIN {X 0,Y 712.276,Z 315.499,A -85,B 0,C 180,E1 33805.547,E2 33805.547} C_VEL
LIN {X 0,Y 712.243,Z 315.502,A -85,B 0,C 180,E1 33802.665,E2 33802.665} C_VEL
LIN {X 0,Y 712.272,Z 315.508,A -85,B 0,C 180,E1 33799.778,E2 33799.778} C_VEL
LIN {X 0,Y 712.25,Z 315.517,A -85,B 0,C 180,E1 33796.868,E2 33796.868} C_VEL
LIN {X 0,Y 713.464,Z 318.858,A -85,B 0,C 180,E1 33796.519,E2 33796.519} C_VEL
LIN {X 0,Y 714.543,Z 321.031,A -85,B 0,C 180,E1 33796.269,E2 33796.269} C_VEL
LIN {X 0,Y 721.038,Z 335.062,A -85,B 0,C 180,E1 33794.736,E2 33794.736} C_VEL
